RoboDK station: Proyecto_Puhueyestewa_Espinoza.rdk

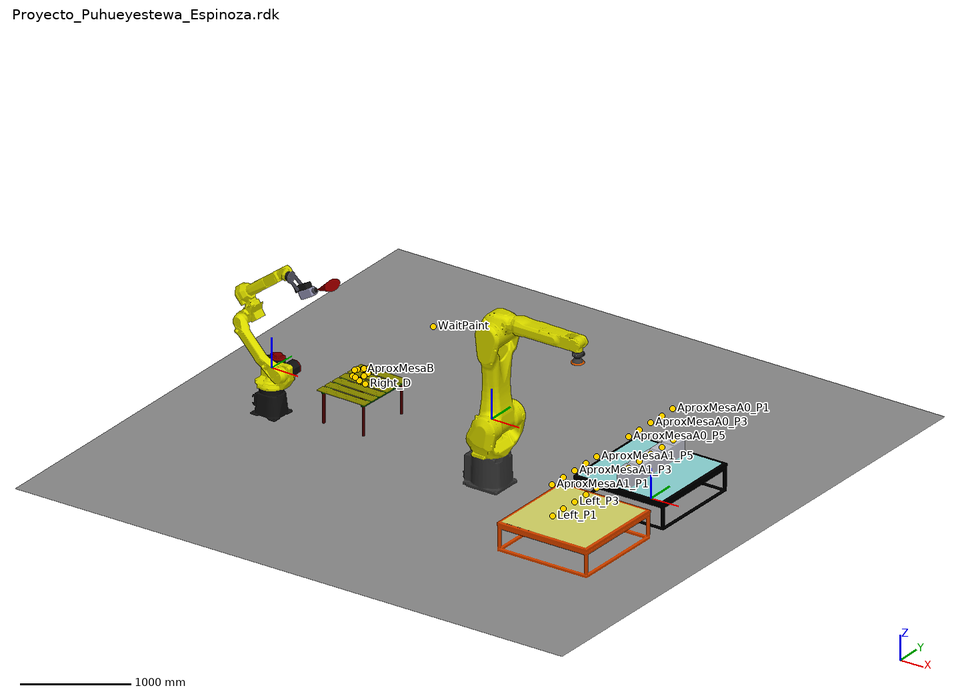
[picture v0: the station drawn from its stored meshes, robots at their saved joint values, targets as dots, program paths as lines]
Station Proyecto_Puhueyestewa_Espinoza (saved by RoboDK 5.3.0). Poses are relative to the parent item; angles as X-Y-Z fixed-axis rotations.
Station parameters (name, value as stored): ColorObject, 3
  - object MesaA1 at (3000, -2200, 0) mm, size 985.8 x 1004.9 x 291.9 mm, geometry from Table-108x114x32-IN.sld
  - object MesaB at (259.9, -1602.19, 600) mm, rotated rx 0 ry 0 rz 88.1 deg, size 656.6 x 530.9 x 335.3 mm, geometry from welding_table.sld
  - frame RobotA Base at (1676.97, -1606.48, 650) mm
    - robot RobotA (model Fanuc M-20iB/25): 6 axes, payload 25 kg, reach 1853 mm, repeatability 0.05 mm, weight 210 kg
        modified DH rows (alpha deg, a mm, theta deg, d mm): 0, 0, 0, 650; -90, 80, -90, 0; 0, 905, 0, 0; -90, 120, 0, 865; 90, 0, 0, 0; -90, 0, 0, 100
        base shift (0, 0, -650) mm
        joint limits [-180, -120, -70, -200, -145, -270] to [180, 120, 230, 200, 145, 270]; home [0, 0, 0, 0, -90, 0]; saved at [0, 0, 0, 0, -90, 180]
      - tool RobotiQ Sanding Kit, TCP at (0, 0, 90.86) mm, size 127 x 139.7 x 103.3 mm
    - target AproxMesaA0_P1 (Cartesian target) at (1323.03, 955.18, 93.07) mm, rotated rx 180 ry 0 rz 0 deg; joints [35.828, 52.673, -25.551, 0, -64.449, -35.828] of RobotA
    - target AproxMesaA0_P2 (Cartesian target) at (1323.03, 780.66, 93.07) mm, rotated rx 180 ry 0 rz 0 deg; joints [30.543, 46.178, -31.005, 0, -58.995, -30.543] of RobotA
    - target AproxMesaA0_P3 (Cartesian target) at (1323.03, 606.48, 93.07) mm, rotated rx -180 ry 0 rz 0 deg; joints [24.627, 41.286, -34.872, 0, -55.128, -24.627] of RobotA
    - target AproxMesaA0_P4 (Cartesian target) at (1323.03, 430.87, 93.07) mm, rotated rx -180 ry 0 rz 0 deg; joints [18.039, 37.651, -37.592, 0, -52.408, -18.039] of RobotA
    - target AproxMesaA0_P5 (Cartesian target) at (1323.03, 257.29, 93.07) mm, rotated rx -180 ry 0 rz 0 deg; joints [11.005, 35.26, -39.302, 0, -50.698, -11.005] of RobotA
    - target AproxMesaA1_P1 (Cartesian target) at (1323.03, -935.11, 93.07) mm, rotated rx -180 ry 0 rz 0 deg; joints [-35.252, 51.823, -26.284, 0, -63.716, 35.252] of RobotA
    - target AproxMesaA1_P2 (Cartesian target) at (1323.03, -761.53, 93.07) mm, rotated rx -180 ry 0 rz 0 deg; joints [-29.925, 45.572, -31.496, 0, -58.504, 29.925] of RobotA
    - target AproxMesaA1_P3 (Cartesian target) at (1323.03, -585.91, 93.07) mm, rotated rx -180 ry 0 rz 0 deg; joints [-23.886, 40.795, -35.247, 0, -54.753, 23.886] of RobotA
    - target AproxMesaA1_P4 (Cartesian target) at (1323.03, -411.74, 93.07) mm, rotated rx -180 ry 0 rz 0 deg; joints [-17.287, 37.329, -37.826, 0, -52.174, 17.287] of RobotA
    - target AproxMesaA1_P5 (Cartesian target) at (1323.03, -237.21, 93.07) mm, rotated rx -180 ry 0 rz 0 deg; joints [-10.165, 35.061, -39.441, 0, -50.559, 10.165] of RobotA
    - target Take_P1 (Cartesian target) at (1323.03, 956.48, -220.35) mm, rotated rx -180 ry 0 rz 0 deg; joints [35.865, 62.489, -38.726, 0, -51.274, -35.865] of RobotA
    - target Take_P2 (Cartesian target) at (1323.03, 780.66, -220.35) mm, rotated rx -180 ry 0 rz 0 deg; joints [30.543, 56.858, -44.792, 0, -45.208, -30.543] of RobotA
    - target Take_P3 (Cartesian target) at (1323.03, 606.48, -220.35) mm, rotated rx -180 ry 0 rz 0 deg; joints [24.627, 52.739, -49.29, 0, -40.71, -24.627] of RobotA
    - target Take_P4 (Cartesian target) at (1323.03, 430.87, -220.35) mm, rotated rx -180 ry 0 rz 0 deg; joints [18.039, 49.747, -52.598, 0, -37.402, -18.039] of RobotA
    - target Take_P5 (Cartesian target) at (1323.03, 257.29, -220.35) mm, rotated rx -180 ry 0 rz 0 deg; joints [11.005, 47.819, -54.753, 0, -35.247, -11.005] of RobotA
    - target Left_P1 (Cartesian target) at (1323.03, -933.81, -220.35) mm, rotated rx -180 ry 0 rz 0 deg; joints [-35.215, 61.659, -39.615, 0, -50.385, 35.215] of RobotA
    - target Left_P2 (Cartesian target) at (1323.03, -760.23, -220.35) mm, rotated rx -180 ry 0 rz 0 deg; joints [-29.882, 56.308, -45.389, 0, -44.611, 29.882] of RobotA
    - target Left_P3 (Cartesian target) at (1323.03, -584.61, -220.35) mm, rotated rx -180 ry 0 rz 0 deg; joints [-23.839, 52.306, -49.766, 0, -40.234, 23.839] of RobotA
    - target Left_P4 (Cartesian target) at (1323.03, -410.44, -220.35) mm, rotated rx -180 ry 0 rz 0 deg; joints [-17.235, 49.468, -52.909, 0, -37.091, 17.235] of RobotA
    - target Left_P5 (Cartesian target) at (1323.03, -235.91, -220.35) mm, rotated rx -180 ry 0 rz 0 deg; joints [-10.11, 47.649, -54.944, 0, -35.056, 10.11] of RobotA
    - target AproxMesaB (Cartesian target) at (-1417.07, 4.29, 103.23) mm, rotated rx 180 ry 0 rz 0 deg; joints [179.826, 38.777, -36.006, 0, -53.994, -179.826] of RobotA
    - target WaitPaint (Cartesian target) at (-643.02, 4.29, 741.53) mm, rotated rx 180 ry 0 rz 0 deg; joints [179.617, -20.046, -8.465, 0, -81.535, -179.617] of RobotA
    - frame MesaA0 Base at (1323.03, 606.48, -660.35) mm
      - object MesaA0 at (0, 0, 0) mm, size 985.8 x 1004.9 x 291.9 mm, geometry from Table-108x114x32-IN.sld
  - frame RobotB Base at (-785.52, -1535.25, 450) mm, rotated rx 0 ry 0 rz -3 deg
    - robot RobotB (model Fanuc M-10iA): 6 axes, payload 10 kg, reach 1420 mm, repeatability 0.08 mm, weight 130 kg
        modified DH rows (alpha deg, a mm, theta deg, d mm): 0, 0, 0, 450; -90, 150, -90, 0; 0, 600, 0, 0; -90, 200, 0, 640; 90, 0, 0, 0; -90, 0, 0, 100
        base shift (0, 0, -450) mm
        joint limits [-180, -90, -95, -190, -190, -360] to [180, 160, 180, 190, 190, 360]; home [0, -44.52, 36.95, 0, -36.95, 0]; saved at [0, -44.52, 36.95, 180, 36.95, 180]
      - tool Paint gun, TCP at (50, 0, 450) mm, rotated rx 0 ry 30 rz 0 deg, size 203.2 x 279.7 x 471.5 mm
    - target Right_D (Cartesian target) at (1128.46, -77.94, 203.78) mm, rotated rx 90 ry -60.18 rz -173.2 deg; joints [-28.769, 42.471, -20.584, -58.905, -97.457, 150.668] of RobotB
    - target Right_M (Cartesian target) at (1071.48, -84.74, 225.06) mm, rotated rx 90 ry -60.18 rz -173.2 deg; joints [-30.393, 36.873, -21.966, -58.048, -98.024, 152.655] of RobotB
    - target Right_U (Cartesian target) at (1002.27, -93, 254.88) mm, rotated rx 90 ry -60.18 rz -173.2 deg; joints [-32.542, 30.646, -22.514, -57, -99.408, 154.203] of RobotB
    - target Center_D (Cartesian target) at (1011.4, -39.87, 300.37) mm, rotated rx 180 ry 0 rz -173.2 deg; joints [-4.924, -0.5, 0.153, -6.683, -60.84, 193.459] of RobotB
    - target Center_M (Cartesian target) at (1050.89, 5.93, 300.37) mm, rotated rx 180 ry 0 rz -173.2 deg; joints [-1.501, 3.048, 0.227, -4.756, -60.572, 189.546] of RobotB
    - target Center_U (Cartesian target) at (1079.26, 49.09, 300.37) mm, rotated rx 180 ry 0 rz -173.2 deg; joints [1.46, 5.834, 0.429, -3.065, -60.572, 186.138] of RobotB
    - target Left_U (Cartesian target) at (1098.26, 69.52, 285.71) mm, rotated rx -90 ry 0 rz -173.2 deg; joints [33.722, 20.618, -41.647, 92.049, -87.698, 138.311] of RobotB
    - target Left_M (Cartesian target) at (1048.72, 63.61, 234.84) mm, rotated rx -90 ry 0 rz -173.2 deg; joints [35.116, 19.049, -47.063, 91.235, -88.851, 132.925] of RobotB
    - target Left_D (Cartesian target) at (1007.9, 58.74, 193.57) mm, rotated rx -90 ry 0 rz -173.2 deg; joints [36.368, 18.195, -51.506, 90.34, -89.729, 128.493] of RobotB
    - target Face_D (Cartesian target) at (972.74, -18.59, 202.79) mm, rotated rx 0 ry -90 rz -173.2 deg; joints [-9.324, -34.09, -22.694, 120.254, 16.17, 246.957] of RobotB
    - target Face_U (Cartesian target) at (973.71, -26.75, 277.71) mm, rotated rx 0 ry -90 rz -173.2 deg; joints [-10.259, -34.141, -16.259, 134.328, 20.806, 232.465] of RobotB
  - Python program Proceso_Industrial (listed below)
  - Python program Estado_Inicial (listed below)
  - object Floor at (1219.35, -1130.77, 0) mm, size 6000 x 6000 x 0 mm, geometry from Floor.sld
  - object Pieza1 at (3000, -650, 429.65) mm, size 150 x 150 x 150 mm, geometry from box.sld
  - object Pieza2 at (3000, -825, 429.65) mm, size 150 x 150 x 150 mm, geometry from box.sld
  - object Pieza3 at (3000, -1000, 429.65) mm, size 150 x 150 x 150 mm, geometry from box.sld
  - object Pieza4 at (3000, -1175, 429.65) mm, size 150 x 150 x 150 mm, geometry from box.sld
  - object Pieza5 at (3000, -1350, 429.65) mm, size 150 x 150 x 150 mm, geometry from box.sld

--- Python program Proceso_Industrial ---
#Laboratorio de Robótica Industrial - Proyecto
#Docente: Ing. María Jose Ramirez Prado
#Integrantes del grupo: Henry Puhueyestewa Sarango - Miguel Espinoza Peña
#Proyecto: Pintado de Objetos
#Paralelo 103

#¬¬¬¬¬¬¬¬¬¬¬¬¬¬¬¬¬¬¬¬¬¬¬¬¬¬¬¬¬¬¬¬¬¬¬¬¬¬¬¬¬¬¬¬¬¬¬¬¬¬¬¬¬¬¬¬¬¬¬¬¬¬¬¬¬¬¬¬¬¬¬¬¬¬¬¬¬¬¬¬¬¬¬¬¬¬¬¬¬¬¬¬¬¬¬¬¬¬¬¬
#ChooseColors¬¬¬¬¬¬¬¬¬¬¬¬¬¬¬¬¬¬¬¬¬¬¬¬¬¬¬¬¬¬¬¬¬¬¬¬¬¬¬¬¬¬¬¬¬¬¬¬¬¬¬¬¬¬¬¬¬¬¬¬¬¬¬¬¬¬¬¬¬¬¬¬¬¬¬¬¬¬¬¬¬¬¬¬¬¬¬¬
#¬¬¬¬¬¬¬¬¬¬¬¬¬¬¬¬¬¬¬¬¬¬¬¬¬¬¬¬¬¬¬¬¬¬¬¬¬¬¬¬¬¬¬¬¬¬¬¬¬¬¬¬¬¬¬¬¬¬¬¬¬¬¬¬¬¬¬¬¬¬¬¬¬¬¬¬¬¬¬¬¬¬¬¬¬¬¬¬¬¬¬¬¬¬¬¬¬¬¬¬
from robolink import *    # API to communicate with RoboDK
from robodk import *      # basic matrix operations

PARAM_COLOR_OBJECT = 'ColorObject'
RDK = Robolink()
color_object = RDK.getParam(PARAM_COLOR_OBJECT)

color_object_input = mbox('Seleccione el color para pintar el objeto: 1. Rojo, 2. Verde, 3. Azul, 4. Rosado', entry=color_object)
if color_object_input:
    RDK.setParam(PARAM_COLOR_OBJECT, color_object_input)
else:
    raise Exception('Operación cancelada por el usuario')

color=int(color_object_input)

#¬¬¬¬¬¬¬¬¬¬¬¬¬¬¬¬¬¬¬¬¬¬¬¬¬¬¬¬¬¬¬¬¬¬¬¬¬¬¬¬¬¬¬¬¬¬¬¬¬¬¬¬¬¬¬¬¬¬¬¬¬¬¬¬¬¬¬¬¬¬¬¬¬¬¬¬¬¬¬¬¬¬¬¬¬¬¬¬¬¬¬¬¬¬¬¬¬¬¬¬
#Asignación de variables y robots¬¬¬¬¬¬¬¬¬¬¬¬¬¬¬¬¬¬¬¬¬¬¬¬¬¬¬¬¬¬¬¬¬¬¬¬¬¬¬¬¬¬¬¬¬¬¬¬¬¬¬¬¬¬¬¬¬¬¬¬¬¬¬¬¬¬¬¬
#¬¬¬¬¬¬¬¬¬¬¬¬¬¬¬¬¬¬¬¬¬¬¬¬¬¬¬¬¬¬¬¬¬¬¬¬¬¬¬¬¬¬¬¬¬¬¬¬¬¬¬¬¬¬¬¬¬¬¬¬¬¬¬¬¬¬¬¬¬¬¬¬¬¬¬¬¬¬¬¬¬¬¬¬¬¬¬¬¬¬¬¬¬¬¬¬¬¬¬¬
#Se asignan variables a los objetos
toola = 'RobotiQ Sanding Kit'
toolb = 'Paint gun'
objecta = 'Pieza1'
objectb = 'Pieza2'
objectc = 'Pieza3'
objectd = 'Pieza4'
objecte = 'Pieza5'
mesa2 = 'MesaB'
mesa3 = 'MesaA1'
gripper1 = RDK.Item(toola, ITEM_TYPE_TOOL)
gripper2 = RDK.Item(toolb, ITEM_TYPE_TOOL)
pi1 = RDK.Item(objecta, ITEM_TYPE_OBJECT)
pi2 = RDK.Item(objectb, ITEM_TYPE_OBJECT)
pi3 = RDK.Item(objectc, ITEM_TYPE_OBJECT)
pi4 = RDK.Item(objectd, ITEM_TYPE_OBJECT)
pi5 = RDK.Item(objecte, ITEM_TYPE_OBJECT)
mesapaint = RDK.Item(mesa2, ITEM_TYPE_OBJECT)
mesafinal = RDK.Item(mesa3, ITEM_TYPE_OBJECT)

#Con respecto a RobotA
robotA = RDK.Item('RobotA',ITEM_TYPE_ROBOT)
if not robotA.Valid():
    quit()
reference = robotA.Parent()
robotA.setPoseFrame(reference)
pose_ref = robotA.Pose()
print(Pose_2_TxyzRxyz(pose_ref))
home_joints = robotA.JointsHome().tolist()

#Con respecto a RobotB
robotB = RDK.Item('RobotB',ITEM_TYPE_ROBOT)
if not robotB.Valid():
    quit()
reference1 = robotB.Parent()
robotB.setPoseFrame(reference1)
pose_ref1 = robotB.Pose()
print(Pose_2_TxyzRxyz(pose_ref1))
home_joints1 = robotB.JointsHome().tolist()

#¬¬¬¬¬¬¬¬¬¬¬¬¬¬¬¬¬¬¬¬¬¬¬¬¬¬¬¬¬¬¬¬¬¬¬¬¬¬¬¬¬¬¬¬¬¬¬¬¬¬¬¬¬¬¬¬¬¬¬¬¬¬¬¬¬¬¬¬¬¬¬¬¬¬¬¬¬¬¬¬¬¬¬¬¬¬¬¬¬¬¬¬¬¬¬¬¬¬¬¬
#Limpio a pintura anterior¬¬¬¬¬¬¬¬¬¬¬¬¬¬¬¬¬¬¬¬¬¬¬¬¬¬¬¬¬¬¬¬¬¬¬¬¬¬¬¬¬¬¬¬¬¬¬¬¬¬¬¬¬¬¬¬¬¬¬¬¬¬¬¬¬¬¬¬¬¬¬¬¬¬¬
#¬¬¬¬¬¬¬¬¬¬¬¬¬¬¬¬¬¬¬¬¬¬¬¬¬¬¬¬¬¬¬¬¬¬¬¬¬¬¬¬¬¬¬¬¬¬¬¬¬¬¬¬¬¬¬¬¬¬¬¬¬¬¬¬¬¬¬¬¬¬¬¬¬¬¬¬¬¬¬¬¬¬¬¬¬¬¬¬¬¬¬¬¬¬¬¬¬¬¬¬
RDK.Spray_Clear()               #Limpio la pintura
pi1.Recolor([0.90,0.91,0.96,1]) #La pieza inicia blanca
pi2.Recolor([0.90,0.91,0.96,1]) #La pieza inicia blanca
pi3.Recolor([0.90,0.91,0.96,1]) #La pieza inicia blanca
pi4.Recolor([0.90,0.91,0.96,1]) #La pieza inicia blanca
pi5.Recolor([0.90,0.91,0.96,1]) #La pieza inicia blanca

#¬¬¬¬¬¬¬¬¬¬¬¬¬¬¬¬¬¬¬¬¬¬¬¬¬¬¬¬¬¬¬¬¬¬¬¬¬¬¬¬¬¬¬¬¬¬¬¬¬¬¬¬¬¬¬¬¬¬¬¬¬¬¬¬¬¬¬¬¬¬¬¬¬¬¬¬¬¬¬¬¬¬¬¬¬¬¬¬¬¬¬¬¬¬¬¬¬¬¬¬
#Process_Pieza1¬¬¬¬¬¬¬¬¬¬¬¬¬¬¬¬¬¬¬¬¬¬¬¬¬¬¬¬¬¬¬¬¬¬¬¬¬¬¬¬¬¬¬¬¬¬¬¬¬¬¬¬¬¬¬¬¬¬¬¬¬¬¬¬¬¬¬¬¬¬¬¬¬¬¬¬¬¬¬¬¬¬¬¬¬¬
#¬¬¬¬¬¬¬¬¬¬¬¬¬¬¬¬¬¬¬¬¬¬¬¬¬¬¬¬¬¬¬¬¬¬¬¬¬¬¬¬¬¬¬¬¬¬¬¬¬¬¬¬¬¬¬¬¬¬¬¬¬¬¬¬¬¬¬¬¬¬¬¬¬¬¬¬¬¬¬¬¬¬¬¬¬¬¬¬¬¬¬¬¬¬¬¬¬¬¬¬
#Tarea Pick and Place en area de trabajo A0
#RobotA se aproxima a MesaA0 para recoger la pieza
aprox=20
a1 = transl(1323.030,955.182,93.068)*roty(pi)
robotA.MoveJ(a1)
robotA.setSpeed(1000)
#RobotA toma la pieza1 de la MesaA0
b1 = transl(1323.030,956.483,-220.350)*roty(pi)
robotA.MoveJ(b1)
robotA.setSpeed(1000)
pi1.setParentStatic(gripper1)
#RobotA lleva la pieza1 cerca de la MesaB
c1=transl(-1417.075,4.293,400.446)*roty(pi)
robotA.MoveJ(c1)
robotA.setSpeed(1000)
#RobotA deja la pieza1 en la MesaB
d1=transl(-1417.075,4.293,100.367)*roty(pi)
robotA.MoveJ(d1)
robotA.setSpeed(1000)
gripper1.DetachAll()
pi1.setParentStatic(mesapaint)
#RobotA se ubica en la posición de espera
e1=transl(-643.019,4.293,741.529)*roty(pi)
robotA.MoveJ(e1)
robotA.setSpeed(1000)
#RobotB se aproxima a MesaB
aprox=20
a02 = xyzrpw_2_pose([951.091,-99.100,515.373,90.000,-60.175,-173.197])
robotB.MoveJ(a02)
robotB.setSpeed(100)

#¬¬¬¬¬¬¬¬¬¬¬¬¬¬¬¬¬¬¬¬¬¬¬¬¬¬¬¬¬¬¬¬¬¬¬¬¬¬¬¬¬¬¬¬¬¬¬¬¬¬¬¬¬¬¬¬¬¬¬¬¬¬¬¬¬¬¬¬¬¬¬¬¬¬¬¬¬¬¬¬¬¬¬¬¬¬¬¬¬¬¬¬¬¬¬¬¬¬¬¬
#SprayOn1¬¬¬¬¬¬¬¬¬¬¬¬¬¬¬¬¬¬¬¬¬¬¬¬¬¬¬¬¬¬¬¬¬¬¬¬¬¬¬¬¬¬¬¬¬¬¬¬¬¬¬¬¬¬¬¬¬¬¬¬¬¬¬¬¬¬¬¬¬¬¬¬¬¬¬¬¬¬¬¬¬¬¬¬¬¬¬¬¬¬¬¬
#¬¬¬¬¬¬¬¬¬¬¬¬¬¬¬¬¬¬¬¬¬¬¬¬¬¬¬¬¬¬¬¬¬¬¬¬¬¬¬¬¬¬¬¬¬¬¬¬¬¬¬¬¬¬¬¬¬¬¬¬¬¬¬¬¬¬¬¬¬¬¬¬¬¬¬¬¬¬¬¬¬¬¬¬¬¬¬¬¬¬¬¬¬¬¬¬¬¬¬¬
Tool_Name = 'Paint gun'
Object_Name = 'Pieza1'

# Define the default action (0 to deactivate, +1 to activate, -1 to clear any spray gun simulation)
# Setting it to None will display a message
ACTION = +1

# quit if we are not in simulation mode
if RDK.RunMode() != RUNMODE_SIMULATE:
    quit()

# Get any previously added spray gun simulations and display statistics (spray on the part vs spray falling out of the part)
info, data = RDK.Spray_GetStats()
if data.size(1) > 0:
    print("Spray gun statistics:")
    print(info)
    print(data.tr())
    RDK.Spray_Clear()

# Check if we are running this program inside another program and passing arguments
import sys
if len(sys.argv) > 1:
    ACTION = int(sys.argv[1])

# If the default ACTION is None, display a message to activate/deactivate the spray gun
if ACTION is None:
    print('Note: This macro can be called as Spray(1) or SprayOn(0)')
    entry = mbox('Turn gun ON or OFF', ('On', '1'), ('Off', '0'))
    if not entry:
        quit()
    ACTION = int(entry)

if ACTION == 0:
    # Turn the gun off
    RDK.Spray_SetState(SPRAY_OFF)

elif ACTION < 0:
    # Clear all spray simulations (same as pressing ESC key)
    RDK.Spray_Clear()

elif ACTION > 0:

    tool = 0    # auto detect active tool
    obj = 0     # auto detect object in active reference frame
    if Tool_Name is not None:
        tool = RDK.Item(Tool_Name, ITEM_TYPE_TOOL)

    if Object_Name is not None:
        obj = RDK.Item(Object_Name, ITEM_TYPE_OBJECT)

    #options_command = "ELLYPSE PROJECT PARTICLE=SPHERE(4,8,1,1,0.5) STEP=8x8 RAND=2" # simulate
    options_command = "PARTICLE=CUBE(10,10,2) STEP=8x8"

    # Another example with a varying rectancular shape
    # define the rectangular volume as p0, pA, pB, colorRGBA (close and far)
    if color == 1:
        close_param = [-90,-117,  0,  90,-117,0,   -90,117,  0,       1,0,0,1]
        far_param   = [-175,-190,200, 175,-190,200,   -175,190,200,   1,0,0,0.2]
        volume = Mat([close_param, far_param])
        RDK.Spray_Add(tool, obj, "RECTANGLE PARTICLE=SPHERE(2,5) STEP=15x15 RAND=3", volume.tr())
        RDK.Spray_SetState(SPRAY_ON)

    if color == 2:
        close_param = [-90,-117,  0,  90,-117,0,   -90,117,  0,       0,1,0,1]
        far_param   = [-175,-190,200, 175,-190,200,   -175,190,200,   1,0,0,0.2]
        volume = Mat([close_param, far_param])
        RDK.Spray_Add(tool, obj, "RECTANGLE PARTICLE=SPHERE(2,5) STEP=15x15 RAND=3", volume.tr())
        RDK.Spray_SetState(SPRAY_ON)

    if color == 3:
        close_param = [-90,-117,  0,  90,-117,0,   -90,117,  0,       0,0,1,1]
        far_param   = [-175,-190,200, 175,-190,200,   -175,190,200,   1,0,0,0.2]
        volume = Mat([close_param, far_param])
        RDK.Spray_Add(tool, obj, "RECTANGLE PARTICLE=SPHERE(2,5) STEP=15x15 RAND=3", volume.tr())
        RDK.Spray_SetState(SPRAY_ON)

    if color == 4:
        close_param = [-90,-117,  0,  90,-117,0,   -90,117,  0,       1,0,1,1]
        far_param   = [-175,-190,200, 175,-190,200,   -175,190,200,   1,0,0,0.2]
        volume = Mat([close_param, far_param])
        RDK.Spray_Add(tool, obj, "RECTANGLE PARTICLE=SPHERE(2,5) STEP=15x15 RAND=3", volume.tr())
        RDK.Spray_SetState(SPRAY_ON)

#¬¬¬¬¬¬¬¬¬¬¬¬¬¬¬¬¬¬¬¬¬¬¬¬¬¬¬¬¬¬¬¬¬¬¬¬¬¬¬¬¬¬¬¬¬¬¬¬¬¬¬¬¬¬¬¬¬¬¬¬¬¬¬¬¬¬¬¬¬¬¬¬¬¬¬¬¬¬¬¬¬¬¬¬¬¬¬¬¬¬¬¬¬¬¬¬¬¬¬¬
#PP1_A¬¬¬¬¬¬¬¬¬¬¬¬¬¬¬¬¬¬¬¬¬¬¬¬¬¬¬¬¬¬¬¬¬¬¬¬¬¬¬¬¬¬¬¬¬¬¬¬¬¬¬¬¬¬¬¬¬¬¬¬¬¬¬¬¬¬¬¬¬¬¬¬¬¬¬¬¬¬¬¬¬¬¬¬¬¬¬¬¬¬¬¬¬¬¬
#¬¬¬¬¬¬¬¬¬¬¬¬¬¬¬¬¬¬¬¬¬¬¬¬¬¬¬¬¬¬¬¬¬¬¬¬¬¬¬¬¬¬¬¬¬¬¬¬¬¬¬¬¬¬¬¬¬¬¬¬¬¬¬¬¬¬¬¬¬¬¬¬¬¬¬¬¬¬¬¬¬¬¬¬¬¬¬¬¬¬¬¬¬¬¬¬¬¬¬¬
#Tarea Pintado en area de trabajo B
#RobotB pinta pieza1, lado derecho
aprox=20
a2 = xyzrpw_2_pose([1128.463,-77.940,203.783,90.000,-60.175,-173.197])
robotB.MoveJ(a2)
robotB.setSpeed(100)
c2 = xyzrpw_2_pose([1071.476,-84.739,225.057,90.000,-60.175,-173.197])
robotB.MoveJ(c2)
robotB.setSpeed(1000)
d2 = xyzrpw_2_pose([1002.267,-92.996,254.878,90.000,-60.175,-173.197])
robotB.MoveJ(d2)
robotB.setSpeed(1000)
#RobotB pinta pieza1, centro
e2 = xyzrpw_2_pose([1011.397,-39.866,300.368,180.000,0.000,-173.197])
robotB.MoveJ(e2)
robotB.setSpeed(1000)
f2 = xyzrpw_2_pose([1050.893,5.934,300.367,180.000,0.000,-173.197])
robotB.MoveJ(f2)
robotB.setSpeed(1000)
g2 = xyzrpw_2_pose([1079.262,49.092,300.367,180.000,0.000,-173.197])
robotB.MoveJ(g2)
robotB.setSpeed(1000)
#RobotB pinta pieza1, lado izquierdo
h2 = xyzrpw_2_pose([1098.260,69.520,285.711,-90.000,0.000,-173.197])
robotB.MoveJ(h2)
robotB.setSpeed(1000)
i2 = xyzrpw_2_pose([1048.722,63.609,234.840,-90.000,0.000,-173.197])
robotB.MoveJ(i2)
robotB.setSpeed(1000)
j2 = xyzrpw_2_pose([1007.902,58.739,193.572,-90.000,0.000,-173.197])
robotB.MoveJ(j2)
robotB.setSpeed(1000)
#RobotB pinta pieza1, frente
k2 = xyzrpw_2_pose([972.738,-18.594,202.789,0.000,-90.000,-173.197])
robotB.MoveJ(k2)
robotB.setSpeed(1000)
l2 = xyzrpw_2_pose([973.710,-26.748,277.710,0.000,-90.000,-173.197])
robotB.MoveJ(l2)
robotB.setSpeed(1000)
#RobotB se mueve a la posición de home
b2 = xyzrpw_2_pose([670.544,0.000,1022.351,0.000,-60.000,-180.000])
robotB.MoveJ(b2)
robotB.setSpeed(100)
#Color
if color == 1:
    pi1.Recolor([1,0,0,1])
if color == 2:
    pi1.Recolor([0,1,0,1])
if color == 3:
    pi1.Recolor([0,0,1,1])
if color == 4:
    pi1.Recolor([1,0,1,1])

#¬¬¬¬¬¬¬¬¬¬¬¬¬¬¬¬¬¬¬¬¬¬¬¬¬¬¬¬¬¬¬¬¬¬¬¬¬¬¬¬¬¬¬¬¬¬¬¬¬¬¬¬¬¬¬¬¬¬¬¬¬¬¬¬¬¬¬¬¬¬¬¬¬¬¬¬¬¬¬¬¬¬¬¬¬¬¬¬¬¬¬¬¬¬¬¬¬¬¬¬
#PP1_B¬¬¬¬¬¬¬¬¬¬¬¬¬¬¬¬¬¬¬¬¬¬¬¬¬¬¬¬¬¬¬¬¬¬¬¬¬¬¬¬¬¬¬¬¬¬¬¬¬¬¬¬¬¬¬¬¬¬¬¬¬¬¬¬¬¬¬¬¬¬¬¬¬¬¬¬¬¬¬¬¬¬¬¬¬¬¬¬¬¬¬¬¬¬¬
#¬¬¬¬¬¬¬¬¬¬¬¬¬¬¬¬¬¬¬¬¬¬¬¬¬¬¬¬¬¬¬¬¬¬¬¬¬¬¬¬¬¬¬¬¬¬¬¬¬¬¬¬¬¬¬¬¬¬¬¬¬¬¬¬¬¬¬¬¬¬¬¬¬¬¬¬¬¬¬¬¬¬¬¬¬¬¬¬¬¬¬¬¬¬¬¬¬¬¬¬
#Tarea Pick and Place en area de trabajo A1
#RobotA toma la pieza1 de la MesaB
a3=transl(-1417.075,4.293,100.367)*roty(pi)
robotA.MoveJ(a3)
robotA.setSpeed(1000)
mesapaint.DetachAll()
pi1.setParentStatic(gripper1)
#RobotA lleva la pieza1 lejos de la MesaB
b3=transl(-1417.075,4.293,400.446)*roty(pi)
robotA.MoveJ(b3)
robotA.setSpeed(1000)
#RobotA lleva la pieza1 entre MesaB y MesaA1
f3=transl(1323.030,955.182,93.068)*roty(pi)
robotA.MoveJ(f3)
robotA.setSpeed(1000)
#RobotA lleva la pieza1 cerca de la MesaA1
c3=transl(1323.030,-935.107,93.068)*roty(pi)
robotA.MoveJ(c3)
robotA.setSpeed(1000)
#RobotA deja la pieza1 en la MesaA1
d3=transl(1323.030,-933.806,-220.350)*roty(pi)
robotA.MoveJ(d3)
robotA.setSpeed(1000)
gripper1.DetachAll()
pi1.setParentStatic(mesafinal)
#RobotA se mueve a la posición de home
e3=transl(945.000,0.000,834.135)*roty(pi)
robotA.MoveJ(e3)
robotA.setSpeed(1000)

#¬¬¬¬¬¬¬¬¬¬¬¬¬¬¬¬¬¬¬¬¬¬¬¬¬¬¬¬¬¬¬¬¬¬¬¬¬¬¬¬¬¬¬¬¬¬¬¬¬¬¬¬¬¬¬¬¬¬¬¬¬¬¬¬¬¬¬¬¬¬¬¬¬¬¬¬¬¬¬¬¬¬¬¬¬¬¬¬¬¬¬¬¬¬¬¬¬¬¬¬
#Process_Pieza2¬¬¬¬¬¬¬¬¬¬¬¬¬¬¬¬¬¬¬¬¬¬¬¬¬¬¬¬¬¬¬¬¬¬¬¬¬¬¬¬¬¬¬¬¬¬¬¬¬¬¬¬¬¬¬¬¬¬¬¬¬¬¬¬¬¬¬¬¬¬¬¬¬¬¬¬¬¬¬¬¬¬¬¬¬¬
#¬¬¬¬¬¬¬¬¬¬¬¬¬¬¬¬¬¬¬¬¬¬¬¬¬¬¬¬¬¬¬¬¬¬¬¬¬¬¬¬¬¬¬¬¬¬¬¬¬¬¬¬¬¬¬¬¬¬¬¬¬¬¬¬¬¬¬¬¬¬¬¬¬¬¬¬¬¬¬¬¬¬¬¬¬¬¬¬¬¬¬¬¬¬¬¬¬¬¬¬
#Tarea Pick and Place en area de trabajo A0
#RobotA se aproxima a MesaA0 para recoger la pieza
aprox=20
a1 = transl(1323.030,780.657,93.068)*roty(pi)      #Se cambia respecto a AproxMesaA0_P________________________
robotA.MoveJ(a1)
robotA.setSpeed(1000)
#RobotA toma la pieza1 de la MesaA0
b1 = transl(1323.030,780.657,-220.350)*roty(pi)    #Se cambia respecto a Take_P________________________
robotA.MoveJ(b1)
robotA.setSpeed(1000)
pi2.setParentStatic(gripper1)                      #Se cambia el pi_____________________________________
#RobotA lleva la pieza1 cerca de la MesaB
c1=transl(-1417.075,4.293,400.446)*roty(pi)
robotA.MoveJ(c1)
robotA.setSpeed(1000)
#RobotA deja la pieza1 en la MesaB
d1=transl(-1417.075,4.293,100.367)*roty(pi)
robotA.MoveJ(d1)
robotA.setSpeed(1000)
gripper1.DetachAll()
pi2.setParentStatic(mesapaint)                     #Se cambia el pi_____________________________________
#RobotA se ubica en la posición de espera
e1=transl(-643.019,4.293,741.529)*roty(pi)
robotA.MoveJ(e1)
robotA.setSpeed(1000)
#RobotB se aproxima a MesaB
aprox=20
a02 = xyzrpw_2_pose([951.091,-99.100,515.373,90.000,-60.175,-173.197])
robotB.MoveJ(a02)
robotB.setSpeed(100)

#¬¬¬¬¬¬¬¬¬¬¬¬¬¬¬¬¬¬¬¬¬¬¬¬¬¬¬¬¬¬¬¬¬¬¬¬¬¬¬¬¬¬¬¬¬¬¬¬¬¬¬¬¬¬¬¬¬¬¬¬¬¬¬¬¬¬¬¬¬¬¬¬¬¬¬¬¬¬¬¬¬¬¬¬¬¬¬¬¬¬¬¬¬¬¬¬¬¬¬¬
#SprayOn2¬¬¬¬¬¬¬¬¬¬¬¬¬¬¬¬¬¬¬¬¬¬¬¬¬¬¬¬¬¬¬¬¬¬¬¬¬¬¬¬¬¬¬¬¬¬¬¬¬¬¬¬¬¬¬¬¬¬¬¬¬¬¬¬¬¬¬¬¬¬¬¬¬¬¬¬¬¬¬¬¬¬¬¬¬¬¬¬¬¬¬¬
#¬¬¬¬¬¬¬¬¬¬¬¬¬¬¬¬¬¬¬¬¬¬¬¬¬¬¬¬¬¬¬¬¬¬¬¬¬¬¬¬¬¬¬¬¬¬¬¬¬¬¬¬¬¬¬¬¬¬¬¬¬¬¬¬¬¬¬¬¬¬¬¬¬¬¬¬¬¬¬¬¬¬¬¬¬¬¬¬¬¬¬¬¬¬¬¬¬¬¬¬
Tool_Name = 'Paint gun'
Object_Name = 'Pieza2'

# Define the default action (0 to deactivate, +1 to activate, -1 to clear any spray gun simulation)
# Setting it to None will display a message
ACTION = +1

# quit if we are not in simulation mode
if RDK.RunMode() != RUNMODE_SIMULATE:
    quit()

# Get any previously added spray gun simulations and display statistics (spray on the part vs spray falling out of the part)
info, data = RDK.Spray_GetStats()
if data.size(1) > 0:
    print("Spray gun statistics:")
    print(info)
    print(data.tr())
    RDK.Spray_Clear()

# Check if we are running this program inside another program and passing arguments
import sys
if len(sys.argv) > 1:
    ACTION = int(sys.argv[1])

# If the default ACTION is None, display a message to activate/deactivate the spray gun
if ACTION is None:
    print('Note: This macro can be called as Spray(1) or SprayOn(0)')
    entry = mbox('Turn gun ON or OFF', ('On', '1'), ('Off', '0'))
    if not entry:
        quit()
    ACTION = int(entry)

if ACTION == 0:
    # Turn the gun off
    RDK.Spray_SetState(SPRAY_OFF)

elif ACTION < 0:
    # Clear all spray simulations (same as pressing ESC key)
    RDK.Spray_Clear()

elif ACTION > 0:

    tool = 0    # auto detect active tool
    obj = 0     # auto detect object in active reference frame
    if Tool_Name is not None:
        tool = RDK.Item(Tool_Name, ITEM_TYPE_TOOL)

    if Object_Name is not None:
        obj = RDK.Item(Object_Name, ITEM_TYPE_OBJECT)

    #options_command = "ELLYPSE PROJECT PARTICLE=SPHERE(4,8,1,1,0.5) STEP=8x8 RAND=2" # simulate
    options_command = "PARTICLE=CUBE(10,10,2) STEP=8x8"

    # Another example with a varying rectancular shape
    # define the rectangular volume as p0, pA, pB, colorRGBA (close and far)
    if color == 1:
        close_param = [-90,-117,  0,  90,-117,0,   -90,117,  0,       1,0,0,1]
        far_param   = [-175,-190,200, 175,-190,200,   -175,190,200,   1,0,0,0.2]
        volume = Mat([close_param, far_param])
        RDK.Spray_Add(tool, obj, "RECTANGLE PARTICLE=SPHERE(2,5) STEP=15x15 RAND=3", volume.tr())
        RDK.Spray_SetState(SPRAY_ON)

    if color == 2:
        close_param = [-90,-117,  0,  90,-117,0,   -90,117,  0,       0,1,0,1]
        far_param   = [-175,-190,200, 175,-190,200,   -175,190,200,   1,0,0,0.2]
        volume = Mat([close_param, far_param])
        RDK.Spray_Add(tool, obj, "RECTANGLE PARTICLE=SPHERE(2,5) STEP=15x15 RAND=3", volume.tr())
        RDK.Spray_SetState(SPRAY_ON)

    if color == 3:
        close_param = [-90,-117,  0,  90,-117,0,   -90,117,  0,       0,0,1,1]
        far_param   = [-175,-190,200, 175,-190,200,   -175,190,200,   1,0,0,0.2]
        volume = Mat([close_param, far_param])
        RDK.Spray_Add(tool, obj, "RECTANGLE PARTICLE=SPHERE(2,5) STEP=15x15 RAND=3", volume.tr())
        RDK.Spray_SetState(SPRAY_ON)

    if color == 4:
        close_param = [-90,-117,  0,  90,-117,0,   -90,117,  0,       1,0,1,1]
        far_param   = [-175,-190,200, 175,-190,200,   -175,190,200,   1,0,0,0.2]
        volume = Mat([close_param, far_param])
        RDK.Spray_Add(tool, obj, "RECTANGLE PARTICLE=SPHERE(2,5) STEP=15x15 RAND=3", volume.tr())
        RDK.Spray_SetState(SPRAY_ON)

#¬¬¬¬¬¬¬¬¬¬¬¬¬¬¬¬¬¬¬¬¬¬¬¬¬¬¬¬¬¬¬¬¬¬¬¬¬¬¬¬¬¬¬¬¬¬¬¬¬¬¬¬¬¬¬¬¬¬¬¬¬¬¬¬¬¬¬¬¬¬¬¬¬¬¬¬¬¬¬¬¬¬¬¬¬¬¬¬¬¬¬¬¬¬¬¬¬¬¬¬
#PP2_A¬¬¬¬¬¬¬¬¬¬¬¬¬¬¬¬¬¬¬¬¬¬¬¬¬¬¬¬¬¬¬¬¬¬¬¬¬¬¬¬¬¬¬¬¬¬¬¬¬¬¬¬¬¬¬¬¬¬¬¬¬¬¬¬¬¬¬¬¬¬¬¬¬¬¬¬¬¬¬¬¬¬¬¬¬¬¬¬¬¬¬¬¬¬¬
#¬¬¬¬¬¬¬¬¬¬¬¬¬¬¬¬¬¬¬¬¬¬¬¬¬¬¬¬¬¬¬¬¬¬¬¬¬¬¬¬¬¬¬¬¬¬¬¬¬¬¬¬¬¬¬¬¬¬¬¬¬¬¬¬¬¬¬¬¬¬¬¬¬¬¬¬¬¬¬¬¬¬¬¬¬¬¬¬¬¬¬¬¬¬¬¬¬¬¬¬
#Tarea Pintado en area de trabajo B
#RobotB pinta pieza1, lado derecho
aprox=20
a2 = xyzrpw_2_pose([1128.463,-77.940,203.783,90.000,-60.175,-173.197])
robotB.MoveJ(a2)
robotB.setSpeed(100)
c2 = xyzrpw_2_pose([1071.476,-84.739,225.057,90.000,-60.175,-173.197])
robotB.MoveJ(c2)
robotB.setSpeed(1000)
d2 = xyzrpw_2_pose([1002.267,-92.996,254.878,90.000,-60.175,-173.197])
robotB.MoveJ(d2)
robotB.setSpeed(1000)
#RobotB pinta pieza1, centro
e2 = xyzrpw_2_pose([1011.397,-39.866,300.368,180.000,0.000,-173.197])
robotB.MoveJ(e2)
robotB.setSpeed(1000)
f2 = xyzrpw_2_pose([1050.893,5.934,300.367,180.000,0.000,-173.197])
robotB.MoveJ(f2)
robotB.setSpeed(1000)
g2 = xyzrpw_2_pose([1079.262,49.092,300.367,180.000,0.000,-173.197])
robotB.MoveJ(g2)
robotB.setSpeed(1000)
#RobotB pinta pieza1, lado izquierdo
h2 = xyzrpw_2_pose([1098.260,69.520,285.711,-90.000,0.000,-173.197])
robotB.MoveJ(h2)
robotB.setSpeed(1000)
i2 = xyzrpw_2_pose([1048.722,63.609,234.840,-90.000,0.000,-173.197])
robotB.MoveJ(i2)
robotB.setSpeed(1000)
j2 = xyzrpw_2_pose([1007.902,58.739,193.572,-90.000,0.000,-173.197])
robotB.MoveJ(j2)
robotB.setSpeed(1000)
#RobotB pinta pieza1, frente
k2 = xyzrpw_2_pose([972.738,-18.594,202.789,0.000,-90.000,-173.197])
robotB.MoveJ(k2)
robotB.setSpeed(1000)
l2 = xyzrpw_2_pose([973.710,-26.748,277.710,0.000,-90.000,-173.197])
robotB.MoveJ(l2)
robotB.setSpeed(1000)
#RobotB se mueve a la posición de home
b2 = xyzrpw_2_pose([670.544,0.000,1022.351,0.000,-60.000,-180.000])
robotB.MoveJ(b2)
robotB.setSpeed(100)
#Color
if color == 1:
    pi2.Recolor([1,0,0,1])
if color == 2:
    pi2.Recolor([0,1,0,1])
if color == 3:
    pi2.Recolor([0,0,1,1])
if color == 4:
    pi2.Recolor([1,0,1,1])

#¬¬¬¬¬¬¬¬¬¬¬¬¬¬¬¬¬¬¬¬¬¬¬¬¬¬¬¬¬¬¬¬¬¬¬¬¬¬¬¬¬¬¬¬¬¬¬¬¬¬¬¬¬¬¬¬¬¬¬¬¬¬¬¬¬¬¬¬¬¬¬¬¬¬¬¬¬¬¬¬¬¬¬¬¬¬¬¬¬¬¬¬¬¬¬¬¬¬¬¬
#PP2_B¬¬¬¬¬¬¬¬¬¬¬¬¬¬¬¬¬¬¬¬¬¬¬¬¬¬¬¬¬¬¬¬¬¬¬¬¬¬¬¬¬¬¬¬¬¬¬¬¬¬¬¬¬¬¬¬¬¬¬¬¬¬¬¬¬¬¬¬¬¬¬¬¬¬¬¬¬¬¬¬¬¬¬¬¬¬¬¬¬¬¬¬¬¬¬
#¬¬¬¬¬¬¬¬¬¬¬¬¬¬¬¬¬¬¬¬¬¬¬¬¬¬¬¬¬¬¬¬¬¬¬¬¬¬¬¬¬¬¬¬¬¬¬¬¬¬¬¬¬¬¬¬¬¬¬¬¬¬¬¬¬¬¬¬¬¬¬¬¬¬¬¬¬¬¬¬¬¬¬¬¬¬¬¬¬¬¬¬¬¬¬¬¬¬¬¬
#Tarea Pick and Place en area de trabajo A1
#RobotA toma la pieza1 de la MesaB
a3=transl(-1417.075,4.293,100.367)*roty(pi)
robotA.MoveJ(a3)
robotA.setSpeed(1000)
mesapaint.DetachAll()
pi2.setParentStatic(gripper1)                          #Se cambia el pi_____________________________________
#RobotA lleva la pieza1 lejos de la MesaB
b3=transl(-1417.075,4.293,400.446)*roty(pi)
robotA.MoveJ(b3)
robotA.setSpeed(1000)
#RobotA lleva la pieza1 entre MesaB y MesaA1
f3=transl(1323.030,780.657,93.068)*roty(pi)            #Se cambia el AproxMesaA0_P_____________________________________
robotA.MoveJ(f3)
robotA.setSpeed(1000)
#RobotA lleva la pieza1 cerca de la MesaA1
c3=transl(1323.030,-761.529,93.068)*roty(pi)           #Se cambia el AproxMesaA1_P__________________________
robotA.MoveJ(c3)
robotA.setSpeed(1000)
#RobotA deja la pieza1 en la MesaA1
d3=transl(1323.030,-760.228,-220.350)*roty(pi)        #Se cambia respecto a Left_P________________________
robotA.MoveJ(d3)
robotA.setSpeed(1000)
gripper1.DetachAll()
pi2.setParentStatic(mesafinal)                        #Se cambia el pi_____________________________________
#RobotA se mueve a la posición de home
e3=transl(945.000,0.000,834.135)*roty(pi)
robotA.MoveJ(e3)
robotA.setSpeed(1000)

#¬¬¬¬¬¬¬¬¬¬¬¬¬¬¬¬¬¬¬¬¬¬¬¬¬¬¬¬¬¬¬¬¬¬¬¬¬¬¬¬¬¬¬¬¬¬¬¬¬¬¬¬¬¬¬¬¬¬¬¬¬¬¬¬¬¬¬¬¬¬¬¬¬¬¬¬¬¬¬¬¬¬¬¬¬¬¬¬¬¬¬¬¬¬¬¬¬¬¬¬
#Process_Pieza3¬¬¬¬¬¬¬¬¬¬¬¬¬¬¬¬¬¬¬¬¬¬¬¬¬¬¬¬¬¬¬¬¬¬¬¬¬¬¬¬¬¬¬¬¬¬¬¬¬¬¬¬¬¬¬¬¬¬¬¬¬¬¬¬¬¬¬¬¬¬¬¬¬¬¬¬¬¬¬¬¬¬¬¬¬¬
#¬¬¬¬¬¬¬¬¬¬¬¬¬¬¬¬¬¬¬¬¬¬¬¬¬¬¬¬¬¬¬¬¬¬¬¬¬¬¬¬¬¬¬¬¬¬¬¬¬¬¬¬¬¬¬¬¬¬¬¬¬¬¬¬¬¬¬¬¬¬¬¬¬¬¬¬¬¬¬¬¬¬¬¬¬¬¬¬¬¬¬¬¬¬¬¬¬¬¬¬
#Tarea Pick and Place en area de trabajo A0
#RobotA se aproxima a MesaA0 para recoger la pieza
aprox=20
a1 = transl(1323.030,606.483,93.068)*roty(pi)      #Se cambia respecto a AproxMesaA0_P________________________
robotA.MoveJ(a1)
robotA.setSpeed(1000)
#RobotA toma la pieza1 de la MesaA0
b1 = transl(1323.030,606.483,-220.350)*roty(pi)    #Se cambia respecto a Take_P________________________
robotA.MoveJ(b1)
robotA.setSpeed(1000)
pi3.setParentStatic(gripper1)                      #Se cambia el pi_____________________________________
#RobotA lleva la pieza1 cerca de la MesaB
c1=transl(-1417.075,4.293,400.446)*roty(pi)
robotA.MoveJ(c1)
robotA.setSpeed(1000)
#RobotA deja la pieza1 en la MesaB
d1=transl(-1417.075,4.293,100.367)*roty(pi)
robotA.MoveJ(d1)
robotA.setSpeed(1000)
gripper1.DetachAll()
pi3.setParentStatic(mesapaint)                     #Se cambia el pi_____________________________________
#RobotA se ubica en la posición de espera
e1=transl(-643.019,4.293,741.529)*roty(pi)
robotA.MoveJ(e1)
robotA.setSpeed(1000)
#RobotB se aproxima a MesaB
aprox=20
a02 = xyzrpw_2_pose([951.091,-99.100,515.373,90.000,-60.175,-173.197])
robotB.MoveJ(a02)
robotB.setSpeed(100)

#¬¬¬¬¬¬¬¬¬¬¬¬¬¬¬¬¬¬¬¬¬¬¬¬¬¬¬¬¬¬¬¬¬¬¬¬¬¬¬¬¬¬¬¬¬¬¬¬¬¬¬¬¬¬¬¬¬¬¬¬¬¬¬¬¬¬¬¬¬¬¬¬¬¬¬¬¬¬¬¬¬¬¬¬¬¬¬¬¬¬¬¬¬¬¬¬¬¬¬¬
#SprayOn3¬¬¬¬¬¬¬¬¬¬¬¬¬¬¬¬¬¬¬¬¬¬¬¬¬¬¬¬¬¬¬¬¬¬¬¬¬¬¬¬¬¬¬¬¬¬¬¬¬¬¬¬¬¬¬¬¬¬¬¬¬¬¬¬¬¬¬¬¬¬¬¬¬¬¬¬¬¬¬¬¬¬¬¬¬¬¬¬¬¬¬¬
#¬¬¬¬¬¬¬¬¬¬¬¬¬¬¬¬¬¬¬¬¬¬¬¬¬¬¬¬¬¬¬¬¬¬¬¬¬¬¬¬¬¬¬¬¬¬¬¬¬¬¬¬¬¬¬¬¬¬¬¬¬¬¬¬¬¬¬¬¬¬¬¬¬¬¬¬¬¬¬¬¬¬¬¬¬¬¬¬¬¬¬¬¬¬¬¬¬¬¬¬
Tool_Name = 'Paint gun'
Object_Name = 'Pieza3'

# Define the default action (0 to deactivate, +1 to activate, -1 to clear any spray gun simulation)
# Setting it to None will display a message
ACTION = +1

# quit if we are not in simulation mode
if RDK.RunMode() != RUNMODE_SIMULATE:
    quit()

# Get any previously added spray gun simulations and display statistics (spray on the part vs spray falling out of the part)
info, data = RDK.Spray_GetStats()
if data.size(1) > 0:
    print("Spray gun statistics:")
    print(info)
    print(data.tr())
    RDK.Spray_Clear()

# Check if we are running this program inside another program and passing arguments
import sys
if len(sys.argv) > 1:
    ACTION = int(sys.argv[1])

# If the default ACTION is None, display a message to activate/deactivate the spray gun
if ACTION is None:
    print('Note: This macro can be called as Spray(1) or SprayOn(0)')
    entry = mbox('Turn gun ON or OFF', ('On', '1'), ('Off', '0'))
    if not entry:
        quit()
    ACTION = int(entry)

if ACTION == 0:
    # Turn the gun off
    RDK.Spray_SetState(SPRAY_OFF)

elif ACTION < 0:
    # Clear all spray simulations (same as pressing ESC key)
    RDK.Spray_Clear()

elif ACTION > 0:

    tool = 0    # auto detect active tool
    obj = 0     # auto detect object in active reference frame
    if Tool_Name is not None:
        tool = RDK.Item(Tool_Name, ITEM_TYPE_TOOL)

    if Object_Name is not None:
        obj = RDK.Item(Object_Name, ITEM_TYPE_OBJECT)

    #options_command = "ELLYPSE PROJECT PARTICLE=SPHERE(4,8,1,1,0.5) STEP=8x8 RAND=2" # simulate
    options_command = "PARTICLE=CUBE(10,10,2) STEP=8x8"

    # Another example with a varying rectancular shape
    # define the rectangular volume as p0, pA, pB, colorRGBA (close and far)
    if color == 1:
        close_param = [-90,-117,  0,  90,-117,0,   -90,117,  0,       1,0,0,1]
        far_param   = [-175,-190,200, 175,-190,200,   -175,190,200,   1,0,0,0.2]
        volume = Mat([close_param, far_param])
        RDK.Spray_Add(tool, obj, "RECTANGLE PARTICLE=SPHERE(2,5) STEP=15x15 RAND=3", volume.tr())
        RDK.Spray_SetState(SPRAY_ON)

    if color == 2:
        close_param = [-90,-117,  0,  90,-117,0,   -90,117,  0,       0,1,0,1]
        far_param   = [-175,-190,200, 175,-190,200,   -175,190,200,   1,0,0,0.2]
        volume = Mat([close_param, far_param])
        RDK.Spray_Add(tool, obj, "RECTANGLE PARTICLE=SPHERE(2,5) STEP=15x15 RAND=3", volume.tr())
        RDK.Spray_SetState(SPRAY_ON)

    if color == 3:
        close_param = [-90,-117,  0,  90,-117,0,   -90,117,  0,       0,0,1,1]
        far_param   = [-175,-190,200, 175,-190,200,   -175,190,200,   1,0,0,0.2]
        volume = Mat([close_param, far_param])
        RDK.Spray_Add(tool, obj, "RECTANGLE PARTICLE=SPHERE(2,5) STEP=15x15 RAND=3", volume.tr())
        RDK.Spray_SetState(SPRAY_ON)

    if color == 4:
        close_param = [-90,-117,  0,  90,-117,0,   -90,117,  0,       1,0,1,1]
        far_param   = [-175,-190,200, 175,-190,200,   -175,190,200,   1,0,0,0.2]
        volume = Mat([close_param, far_param])
        RDK.Spray_Add(tool, obj, "RECTANGLE PARTICLE=SPHERE(2,5) STEP=15x15 RAND=3", volume.tr())
        RDK.Spray_SetState(SPRAY_ON)

#¬¬¬¬¬¬¬¬¬¬¬¬¬¬¬¬¬¬¬¬¬¬¬¬¬¬¬¬¬¬¬¬¬¬¬¬¬¬¬¬¬¬¬¬¬¬¬¬¬¬¬¬¬¬¬¬¬¬¬¬¬¬¬¬¬¬¬¬¬¬¬¬¬¬¬¬¬¬¬¬¬¬¬¬¬¬¬¬¬¬¬¬¬¬¬¬¬¬¬¬
#PP3_A¬¬¬¬¬¬¬¬¬¬¬¬¬¬¬¬¬¬¬¬¬¬¬¬¬¬¬¬¬¬¬¬¬¬¬¬¬¬¬¬¬¬¬¬¬¬¬¬¬¬¬¬¬¬¬¬¬¬¬¬¬¬¬¬¬¬¬¬¬¬¬¬¬¬¬¬¬¬¬¬¬¬¬¬¬¬¬¬¬¬¬¬¬¬¬
#¬¬¬¬¬¬¬¬¬¬¬¬¬¬¬¬¬¬¬¬¬¬¬¬¬¬¬¬¬¬¬¬¬¬¬¬¬¬¬¬¬¬¬¬¬¬¬¬¬¬¬¬¬¬¬¬¬¬¬¬¬¬¬¬¬¬¬¬¬¬¬¬¬¬¬¬¬¬¬¬¬¬¬¬¬¬¬¬¬¬¬¬¬¬¬¬¬¬¬¬
#Tarea Pintado en area de trabajo B
#RobotB pinta pieza1, lado derecho
aprox=20
a2 = xyzrpw_2_pose([1128.463,-77.940,203.783,90.000,-60.175,-173.197])
robotB.MoveJ(a2)
robotB.setSpeed(100)
c2 = xyzrpw_2_pose([1071.476,-84.739,225.057,90.000,-60.175,-173.197])
robotB.MoveJ(c2)
robotB.setSpeed(1000)
d2 = xyzrpw_2_pose([1002.267,-92.996,254.878,90.000,-60.175,-173.197])
robotB.MoveJ(d2)
robotB.setSpeed(1000)
#RobotB pinta pieza1, centro
e2 = xyzrpw_2_pose([1011.397,-39.866,300.368,180.000,0.000,-173.197])
robotB.MoveJ(e2)
robotB.setSpeed(1000)
f2 = xyzrpw_2_pose([1050.893,5.934,300.367,180.000,0.000,-173.197])
robotB.MoveJ(f2)
robotB.setSpeed(1000)
g2 = xyzrpw_2_pose([1079.262,49.092,300.367,180.000,0.000,-173.197])
robotB.MoveJ(g2)
robotB.setSpeed(1000)
#RobotB pinta pieza1, lado izquierdo
h2 = xyzrpw_2_pose([1098.260,69.520,285.711,-90.000,0.000,-173.197])
robotB.MoveJ(h2)
robotB.setSpeed(1000)
i2 = xyzrpw_2_pose([1048.722,63.609,234.840,-90.000,0.000,-173.197])
robotB.MoveJ(i2)
robotB.setSpeed(1000)
j2 = xyzrpw_2_pose([1007.902,58.739,193.572,-90.000,0.000,-173.197])
robotB.MoveJ(j2)
robotB.setSpeed(1000)
#RobotB pinta pieza1, frente
k2 = xyzrpw_2_pose([972.738,-18.594,202.789,0.000,-90.000,-173.197])
robotB.MoveJ(k2)
robotB.setSpeed(1000)
l2 = xyzrpw_2_pose([973.710,-26.748,277.710,0.000,-90.000,-173.197])
robotB.MoveJ(l2)
robotB.setSpeed(1000)
#RobotB se mueve a la posición de home
b2 = xyzrpw_2_pose([670.544,0.000,1022.351,0.000,-60.000,-180.000])
robotB.MoveJ(b2)
robotB.setSpeed(100)
#Color
if color == 1:
    pi3.Recolor([1,0,0,1])
if color == 2:
    pi3.Recolor([0,1,0,1])
if color == 3:
    pi3.Recolor([0,0,1,1])
if color == 4:
    pi3.Recolor([1,0,1,1])

#¬¬¬¬¬¬¬¬¬¬¬¬¬¬¬¬¬¬¬¬¬¬¬¬¬¬¬¬¬¬¬¬¬¬¬¬¬¬¬¬¬¬¬¬¬¬¬¬¬¬¬¬¬¬¬¬¬¬¬¬¬¬¬¬¬¬¬¬¬¬¬¬¬¬¬¬¬¬¬¬¬¬¬¬¬¬¬¬¬¬¬¬¬¬¬¬¬¬¬¬
#PP3_B¬¬¬¬¬¬¬¬¬¬¬¬¬¬¬¬¬¬¬¬¬¬¬¬¬¬¬¬¬¬¬¬¬¬¬¬¬¬¬¬¬¬¬¬¬¬¬¬¬¬¬¬¬¬¬¬¬¬¬¬¬¬¬¬¬¬¬¬¬¬¬¬¬¬¬¬¬¬¬¬¬¬¬¬¬¬¬¬¬¬¬¬¬¬¬
#¬¬¬¬¬¬¬¬¬¬¬¬¬¬¬¬¬¬¬¬¬¬¬¬¬¬¬¬¬¬¬¬¬¬¬¬¬¬¬¬¬¬¬¬¬¬¬¬¬¬¬¬¬¬¬¬¬¬¬¬¬¬¬¬¬¬¬¬¬¬¬¬¬¬¬¬¬¬¬¬¬¬¬¬¬¬¬¬¬¬¬¬¬¬¬¬¬¬¬¬
#Tarea Pick and Place en area de trabajo A1
#RobotA toma la pieza1 de la MesaB
a3=transl(-1417.075,4.293,100.367)*roty(pi)
robotA.MoveJ(a3)
robotA.setSpeed(1000)
mesapaint.DetachAll()
pi3.setParentStatic(gripper1)                          #Se cambia el pi_____________________________________
#RobotA lleva la pieza1 lejos de la MesaB
b3=transl(-1417.075,4.293,400.446)*roty(pi)
robotA.MoveJ(b3)
robotA.setSpeed(1000)
#RobotA lleva la pieza1 entre MesaB y MesaA1
f3=transl(1323.030,606.483,93.068)*roty(pi)            #Se cambia el AproxMesaA0_P_____________________________________
robotA.MoveJ(f3)
robotA.setSpeed(1000)
#RobotA lleva la pieza1 cerca de la MesaA1
c3=transl(1323.030,-585.913,93.068)*roty(pi)           #Se cambia el AproxMesaA1_P__________________________
robotA.MoveJ(c3)
robotA.setSpeed(1000)
#RobotA deja la pieza1 en la MesaA1
d3=transl(1323.030,-584.612,-220.350)*roty(pi)        #Se cambia respecto a Left_P________________________
robotA.MoveJ(d3)
robotA.setSpeed(1000)
gripper1.DetachAll()
pi3.setParentStatic(mesafinal)                        #Se cambia el pi_____________________________________
#RobotA se mueve a la posición de home
e3=transl(945.000,0.000,834.135)*roty(pi)
robotA.MoveJ(e3)
robotA.setSpeed(1000)

#¬¬¬¬¬¬¬¬¬¬¬¬¬¬¬¬¬¬¬¬¬¬¬¬¬¬¬¬¬¬¬¬¬¬¬¬¬¬¬¬¬¬¬¬¬¬¬¬¬¬¬¬¬¬¬¬¬¬¬¬¬¬¬¬¬¬¬¬¬¬¬¬¬¬¬¬¬¬¬¬¬¬¬¬¬¬¬¬¬¬¬¬¬¬¬¬¬¬¬¬
#Process_Pieza4¬¬¬¬¬¬¬¬¬¬¬¬¬¬¬¬¬¬¬¬¬¬¬¬¬¬¬¬¬¬¬¬¬¬¬¬¬¬¬¬¬¬¬¬¬¬¬¬¬¬¬¬¬¬¬¬¬¬¬¬¬¬¬¬¬¬¬¬¬¬¬¬¬¬¬¬¬¬¬¬¬¬¬¬¬¬
#¬¬¬¬¬¬¬¬¬¬¬¬¬¬¬¬¬¬¬¬¬¬¬¬¬¬¬¬¬¬¬¬¬¬¬¬¬¬¬¬¬¬¬¬¬¬¬¬¬¬¬¬¬¬¬¬¬¬¬¬¬¬¬¬¬¬¬¬¬¬¬¬¬¬¬¬¬¬¬¬¬¬¬¬¬¬¬¬¬¬¬¬¬¬¬¬¬¬¬¬
#Tarea Pick and Place en area de trabajo A0
#RobotA se aproxima a MesaA0 para recoger la pieza
aprox=20
a1 = transl(1323.030,430.867,93.068)*roty(pi)      #Se cambia respecto a AproxMesaA0_P________________________
robotA.MoveJ(a1)
robotA.setSpeed(1000)
#RobotA toma la pieza1 de la MesaA0
b1 = transl(1323.030,430.867,-220.350)*roty(pi)    #Se cambia respecto a Take_P________________________
robotA.MoveJ(b1)
robotA.setSpeed(1000)
pi4.setParentStatic(gripper1)                      #Se cambia el pi_____________________________________
#RobotA lleva la pieza1 cerca de la MesaB
c1=transl(-1417.075,4.293,400.446)*roty(pi)
robotA.MoveJ(c1)
robotA.setSpeed(1000)
#RobotA deja la pieza1 en la MesaB
d1=transl(-1417.075,4.293,100.367)*roty(pi)
robotA.MoveJ(d1)
robotA.setSpeed(1000)
gripper1.DetachAll()
pi4.setParentStatic(mesapaint)                     #Se cambia el pi_____________________________________
#RobotA se ubica en la posición de espera
e1=transl(-643.019,4.293,741.529)*roty(pi)
robotA.MoveJ(e1)
robotA.setSpeed(1000)
#RobotB se aproxima a MesaB
aprox=20
a02 = xyzrpw_2_pose([951.091,-99.100,515.373,90.000,-60.175,-173.197])
robotB.MoveJ(a02)
robotB.setSpeed(100)

#¬¬¬¬¬¬¬¬¬¬¬¬¬¬¬¬¬¬¬¬¬¬¬¬¬¬¬¬¬¬¬¬¬¬¬¬¬¬¬¬¬¬¬¬¬¬¬¬¬¬¬¬¬¬¬¬¬¬¬¬¬¬¬¬¬¬¬¬¬¬¬¬¬¬¬¬¬¬¬¬¬¬¬¬¬¬¬¬¬¬¬¬¬¬¬¬¬¬¬¬
#SprayOn4¬¬¬¬¬¬¬¬¬¬¬¬¬¬¬¬¬¬¬¬¬¬¬¬¬¬¬¬¬¬¬¬¬¬¬¬¬¬¬¬¬¬¬¬¬¬¬¬¬¬¬¬¬¬¬¬¬¬¬¬¬¬¬¬¬¬¬¬¬¬¬¬¬¬¬¬¬¬¬¬¬¬¬¬¬¬¬¬¬¬¬¬
#¬¬¬¬¬¬¬¬¬¬¬¬¬¬¬¬¬¬¬¬¬¬¬¬¬¬¬¬¬¬¬¬¬¬¬¬¬¬¬¬¬¬¬¬¬¬¬¬¬¬¬¬¬¬¬¬¬¬¬¬¬¬¬¬¬¬¬¬¬¬¬¬¬¬¬¬¬¬¬¬¬¬¬¬¬¬¬¬¬¬¬¬¬¬¬¬¬¬¬¬
Tool_Name = 'Paint gun'
Object_Name = 'Pieza4'

# Define the default action (0 to deactivate, +1 to activate, -1 to clear any spray gun simulation)
# Setting it to None will display a message
ACTION = +1

# quit if we are not in simulation mode
if RDK.RunMode() != RUNMODE_SIMULATE:
    quit()

# Get any previously added spray gun simulations and display statistics (spray on the part vs spray falling out of the part)
info, data = RDK.Spray_GetStats()
if data.size(1) > 0:
    print("Spray gun statistics:")
    print(info)
    print(data.tr())
    RDK.Spray_Clear()

# Check if we are running this program inside another program and passing arguments
import sys
if len(sys.argv) > 1:
    ACTION = int(sys.argv[1])

# If the default ACTION is None, display a message to activate/deactivate the spray gun
if ACTION is None:
    print('Note: This macro can be called as Spray(1) or SprayOn(0)')
    entry = mbox('Turn gun ON or OFF', ('On', '1'), ('Off', '0'))
    if not entry:
        quit()
    ACTION = int(entry)

if ACTION == 0:
    # Turn the gun off
    RDK.Spray_SetState(SPRAY_OFF)

elif ACTION < 0:
    # Clear all spray simulations (same as pressing ESC key)
    RDK.Spray_Clear()

elif ACTION > 0:

    tool = 0    # auto detect active tool
    obj = 0     # auto detect object in active reference frame
    if Tool_Name is not None:
        tool = RDK.Item(Tool_Name, ITEM_TYPE_TOOL)

    if Object_Name is not None:
        obj = RDK.Item(Object_Name, ITEM_TYPE_OBJECT)

    #options_command = "ELLYPSE PROJECT PARTICLE=SPHERE(4,8,1,1,0.5) STEP=8x8 RAND=2" # simulate
    options_command = "PARTICLE=CUBE(10,10,2) STEP=8x8"

    # Another example with a varying rectancular shape
    # define the rectangular volume as p0, pA, pB, colorRGBA (close and far)
    if color == 1:
        close_param = [-90,-117,  0,  90,-117,0,   -90,117,  0,       1,0,0,1]
        far_param   = [-175,-190,200, 175,-190,200,   -175,190,200,   1,0,0,0.2]
        volume = Mat([close_param, far_param])
        RDK.Spray_Add(tool, obj, "RECTANGLE PARTICLE=SPHERE(2,5) STEP=15x15 RAND=3", volume.tr())
        RDK.Spray_SetState(SPRAY_ON)

    if color == 2:
        close_param = [-90,-117,  0,  90,-117,0,   -90,117,  0,       0,1,0,1]
        far_param   = [-175,-190,200, 175,-190,200,   -175,190,200,   1,0,0,0.2]
        volume = Mat([close_param, far_param])
        RDK.Spray_Add(tool, obj, "RECTANGLE PARTICLE=SPHERE(2,5) STEP=15x15 RAND=3", volume.tr())
        RDK.Spray_SetState(SPRAY_ON)

    if color == 3:
        close_param = [-90,-117,  0,  90,-117,0,   -90,117,  0,       0,0,1,1]
        far_param   = [-175,-190,200, 175,-190,200,   -175,190,200,   1,0,0,0.2]
        volume = Mat([close_param, far_param])
        RDK.Spray_Add(tool, obj, "RECTANGLE PARTICLE=SPHERE(2,5) STEP=15x15 RAND=3", volume.tr())
        RDK.Spray_SetState(SPRAY_ON)

    if color == 4:
        close_param = [-90,-117,  0,  90,-117,0,   -90,117,  0,       1,0,1,1]
        far_param   = [-175,-190,200, 175,-190,200,   -175,190,200,   1,0,0,0.2]
        volume = Mat([close_param, far_param])
        RDK.Spray_Add(tool, obj, "RECTANGLE PARTICLE=SPHERE(2,5) STEP=15x15 RAND=3", volume.tr())
        RDK.Spray_SetState(SPRAY_ON)

#¬¬¬¬¬¬¬¬¬¬¬¬¬¬¬¬¬¬¬¬¬¬¬¬¬¬¬¬¬¬¬¬¬¬¬¬¬¬¬¬¬¬¬¬¬¬¬¬¬¬¬¬¬¬¬¬¬¬¬¬¬¬¬¬¬¬¬¬¬¬¬¬¬¬¬¬¬¬¬¬¬¬¬¬¬¬¬¬¬¬¬¬¬¬¬¬¬¬¬¬
#PP4_A¬¬¬¬¬¬¬¬¬¬¬¬¬¬¬¬¬¬¬¬¬¬¬¬¬¬¬¬¬¬¬¬¬¬¬¬¬¬¬¬¬¬¬¬¬¬¬¬¬¬¬¬¬¬¬¬¬¬¬¬¬¬¬¬¬¬¬¬¬¬¬¬¬¬¬¬¬¬¬¬¬¬¬¬¬¬¬¬¬¬¬¬¬¬¬
#¬¬¬¬¬¬¬¬¬¬¬¬¬¬¬¬¬¬¬¬¬¬¬¬¬¬¬¬¬¬¬¬¬¬¬¬¬¬¬¬¬¬¬¬¬¬¬¬¬¬¬¬¬¬¬¬¬¬¬¬¬¬¬¬¬¬¬¬¬¬¬¬¬¬¬¬¬¬¬¬¬¬¬¬¬¬¬¬¬¬¬¬¬¬¬¬¬¬¬¬
#Tarea Pintado en area de trabajo B
#RobotB pinta pieza1, lado derecho
aprox=20
a2 = xyzrpw_2_pose([1128.463,-77.940,203.783,90.000,-60.175,-173.197])
robotB.MoveJ(a2)
robotB.setSpeed(100)
c2 = xyzrpw_2_pose([1071.476,-84.739,225.057,90.000,-60.175,-173.197])
robotB.MoveJ(c2)
robotB.setSpeed(1000)
d2 = xyzrpw_2_pose([1002.267,-92.996,254.878,90.000,-60.175,-173.197])
robotB.MoveJ(d2)
robotB.setSpeed(1000)
#RobotB pinta pieza1, centro
e2 = xyzrpw_2_pose([1011.397,-39.866,300.368,180.000,0.000,-173.197])
robotB.MoveJ(e2)
robotB.setSpeed(1000)
f2 = xyzrpw_2_pose([1050.893,5.934,300.367,180.000,0.000,-173.197])
robotB.MoveJ(f2)
robotB.setSpeed(1000)
g2 = xyzrpw_2_pose([1079.262,49.092,300.367,180.000,0.000,-173.197])
robotB.MoveJ(g2)
robotB.setSpeed(1000)
#RobotB pinta pieza1, lado izquierdo
h2 = xyzrpw_2_pose([1098.260,69.520,285.711,-90.000,0.000,-173.197])
robotB.MoveJ(h2)
robotB.setSpeed(1000)
i2 = xyzrpw_2_pose([1048.722,63.609,234.840,-90.000,0.000,-173.197])
robotB.MoveJ(i2)
robotB.setSpeed(1000)
j2 = xyzrpw_2_pose([1007.902,58.739,193.572,-90.000,0.000,-173.197])
robotB.MoveJ(j2)
robotB.setSpeed(1000)
#RobotB pinta pieza1, frente
k2 = xyzrpw_2_pose([972.738,-18.594,202.789,0.000,-90.000,-173.197])
robotB.MoveJ(k2)
robotB.setSpeed(1000)
l2 = xyzrpw_2_pose([973.710,-26.748,277.710,0.000,-90.000,-173.197])
robotB.MoveJ(l2)
robotB.setSpeed(1000)
#RobotB se mueve a la posición de home
b2 = xyzrpw_2_pose([670.544,0.000,1022.351,0.000,-60.000,-180.000])
robotB.MoveJ(b2)
robotB.setSpeed(100)
#Color
if color == 1:
    pi4.Recolor([1,0,0,1])
if color == 2:
    pi4.Recolor([0,1,0,1])
if color == 3:
    pi4.Recolor([0,0,1,1])
if color == 4:
    pi4.Recolor([1,0,1,1])

#¬¬¬¬¬¬¬¬¬¬¬¬¬¬¬¬¬¬¬¬¬¬¬¬¬¬¬¬¬¬¬¬¬¬¬¬¬¬¬¬¬¬¬¬¬¬¬¬¬¬¬¬¬¬¬¬¬¬¬¬¬¬¬¬¬¬¬¬¬¬¬¬¬¬¬¬¬¬¬¬¬¬¬¬¬¬¬¬¬¬¬¬¬¬¬¬¬¬¬¬
#PP4_B¬¬¬¬¬¬¬¬¬¬¬¬¬¬¬¬¬¬¬¬¬¬¬¬¬¬¬¬¬¬¬¬¬¬¬¬¬¬¬¬¬¬¬¬¬¬¬¬¬¬¬¬¬¬¬¬¬¬¬¬¬¬¬¬¬¬¬¬¬¬¬¬¬¬¬¬¬¬¬¬¬¬¬¬¬¬¬¬¬¬¬¬¬¬¬
#¬¬¬¬¬¬¬¬¬¬¬¬¬¬¬¬¬¬¬¬¬¬¬¬¬¬¬¬¬¬¬¬¬¬¬¬¬¬¬¬¬¬¬¬¬¬¬¬¬¬¬¬¬¬¬¬¬¬¬¬¬¬¬¬¬¬¬¬¬¬¬¬¬¬¬¬¬¬¬¬¬¬¬¬¬¬¬¬¬¬¬¬¬¬¬¬¬¬¬¬
#Tarea Pick and Place en area de trabajo A1
#RobotA toma la pieza1 de la MesaB
a3=transl(-1417.075,4.293,100.367)*roty(pi)
robotA.MoveJ(a3)
robotA.setSpeed(1000)
mesapaint.DetachAll()
pi4.setParentStatic(gripper1)                          #Se cambia el pi_____________________________________
#RobotA lleva la pieza1 lejos de la MesaB
b3=transl(-1417.075,4.293,400.446)*roty(pi)
robotA.MoveJ(b3)
robotA.setSpeed(1000)
#RobotA lleva la pieza1 entre MesaB y MesaA1
f3=transl(1323.030,430.867,93.068)*roty(pi)            #Se cambia el AproxMesaA0_P_____________________________________
robotA.MoveJ(f3)
robotA.setSpeed(1000)
#RobotA lleva la pieza1 cerca de la MesaA1
c3=transl(1323.030,-411.739,93.068)*roty(pi)           #Se cambia el AproxMesaA1_P__________________________
robotA.MoveJ(c3)
robotA.setSpeed(1000)
#RobotA deja la pieza1 en la MesaA1
d3=transl(1323.030,-410.438,-220.350)*roty(pi)        #Se cambia respecto a Left_P________________________
robotA.MoveJ(d3)
robotA.setSpeed(1000)
gripper1.DetachAll()
pi4.setParentStatic(mesafinal)                        #Se cambia el pi_____________________________________
#RobotA se mueve a la posición de home
e3=transl(945.000,0.000,834.135)*roty(pi)
robotA.MoveJ(e3)
robotA.setSpeed(1000)

#¬¬¬¬¬¬¬¬¬¬¬¬¬¬¬¬¬¬¬¬¬¬¬¬¬¬¬¬¬¬¬¬¬¬¬¬¬¬¬¬¬¬¬¬¬¬¬¬¬¬¬¬¬¬¬¬¬¬¬¬¬¬¬¬¬¬¬¬¬¬¬¬¬¬¬¬¬¬¬¬¬¬¬¬¬¬¬¬¬¬¬¬¬¬¬¬¬¬¬¬
#Process_Pieza5¬¬¬¬¬¬¬¬¬¬¬¬¬¬¬¬¬¬¬¬¬¬¬¬¬¬¬¬¬¬¬¬¬¬¬¬¬¬¬¬¬¬¬¬¬¬¬¬¬¬¬¬¬¬¬¬¬¬¬¬¬¬¬¬¬¬¬¬¬¬¬¬¬¬¬¬¬¬¬¬¬¬¬¬¬¬
#¬¬¬¬¬¬¬¬¬¬¬¬¬¬¬¬¬¬¬¬¬¬¬¬¬¬¬¬¬¬¬¬¬¬¬¬¬¬¬¬¬¬¬¬¬¬¬¬¬¬¬¬¬¬¬¬¬¬¬¬¬¬¬¬¬¬¬¬¬¬¬¬¬¬¬¬¬¬¬¬¬¬¬¬¬¬¬¬¬¬¬¬¬¬¬¬¬¬¬¬
#Tarea Pick and Place en area de trabajo A0
#RobotA se aproxima a MesaA0 para recoger la pieza
aprox=20
a1 = transl(1323.030,257.289,93.068)*roty(pi)      #Se cambia respecto a AproxMesaA0_P________________________
robotA.MoveJ(a1)
robotA.setSpeed(1000)
#RobotA toma la pieza1 de la MesaA0
b1 = transl(1323.030,257.289,-220.350)*roty(pi)    #Se cambia respecto a Take_P________________________
robotA.MoveJ(b1)
robotA.setSpeed(1000)
pi5.setParentStatic(gripper1)                      #Se cambia el pi_____________________________________
#RobotA lleva la pieza1 cerca de la MesaB
c1=transl(-1417.075,4.293,400.446)*roty(pi)
robotA.MoveJ(c1)
robotA.setSpeed(1000)
#RobotA deja la pieza1 en la MesaB
d1=transl(-1417.075,4.293,100.367)*roty(pi)
robotA.MoveJ(d1)
robotA.setSpeed(1000)
gripper1.DetachAll()
pi5.setParentStatic(mesapaint)                     #Se cambia el pi_____________________________________
#RobotA se ubica en la posición de espera
e1=transl(-643.019,4.293,741.529)*roty(pi)
robotA.MoveJ(e1)
robotA.setSpeed(1000)
#RobotB se aproxima a MesaB
aprox=20
a02 = xyzrpw_2_pose([951.091,-99.100,515.373,90.000,-60.175,-173.197])
robotB.MoveJ(a02)
robotB.setSpeed(100)

#¬¬¬¬¬¬¬¬¬¬¬¬¬¬¬¬¬¬¬¬¬¬¬¬¬¬¬¬¬¬¬¬¬¬¬¬¬¬¬¬¬¬¬¬¬¬¬¬¬¬¬¬¬¬¬¬¬¬¬¬¬¬¬¬¬¬¬¬¬¬¬¬¬¬¬¬¬¬¬¬¬¬¬¬¬¬¬¬¬¬¬¬¬¬¬¬¬¬¬¬
#SprayOn5¬¬¬¬¬¬¬¬¬¬¬¬¬¬¬¬¬¬¬¬¬¬¬¬¬¬¬¬¬¬¬¬¬¬¬¬¬¬¬¬¬¬¬¬¬¬¬¬¬¬¬¬¬¬¬¬¬¬¬¬¬¬¬¬¬¬¬¬¬¬¬¬¬¬¬¬¬¬¬¬¬¬¬¬¬¬¬¬¬¬¬¬
#¬¬¬¬¬¬¬¬¬¬¬¬¬¬¬¬¬¬¬¬¬¬¬¬¬¬¬¬¬¬¬¬¬¬¬¬¬¬¬¬¬¬¬¬¬¬¬¬¬¬¬¬¬¬¬¬¬¬¬¬¬¬¬¬¬¬¬¬¬¬¬¬¬¬¬¬¬¬¬¬¬¬¬¬¬¬¬¬¬¬¬¬¬¬¬¬¬¬¬¬
Tool_Name = 'Paint gun'
Object_Name = 'Pieza5'

# Define the default action (0 to deactivate, +1 to activate, -1 to clear any spray gun simulation)
# Setting it to None will display a message
ACTION = +1

# quit if we are not in simulation mode
if RDK.RunMode() != RUNMODE_SIMULATE:
    quit()

# Get any previously added spray gun simulations and display statistics (spray on the part vs spray falling out of the part)
info, data = RDK.Spray_GetStats()
if data.size(1) > 0:
    print("Spray gun statistics:")
    print(info)
    print(data.tr())
    RDK.Spray_Clear()

# Check if we are running this program inside another program and passing arguments
import sys
if len(sys.argv) > 1:
    ACTION = int(sys.argv[1])

# If the default ACTION is None, display a message to activate/deactivate the spray gun
if ACTION is None:
    print('Note: This macro can be called as Spray(1) or SprayOn(0)')
    entry = mbox('Turn gun ON or OFF', ('On', '1'), ('Off', '0'))
    if not entry:
        quit()
    ACTION = int(entry)

if ACTION == 0:
    # Turn the gun off
    RDK.Spray_SetState(SPRAY_OFF)

elif ACTION < 0:
    # Clear all spray simulations (same as pressing ESC key)
    RDK.Spray_Clear()

elif ACTION > 0:

    tool = 0    # auto detect active tool
    obj = 0     # auto detect object in active reference frame
    if Tool_Name is not None:
        tool = RDK.Item(Tool_Name, ITEM_TYPE_TOOL)

    if Object_Name is not None:
        obj = RDK.Item(Object_Name, ITEM_TYPE_OBJECT)

    #options_command = "ELLYPSE PROJECT PARTICLE=SPHERE(4,8,1,1,0.5) STEP=8x8 RAND=2" # simulate
    options_command = "PARTICLE=CUBE(10,10,2) STEP=8x8"

    # Another example with a varying rectancular shape
    # define the rectangular volume as p0, pA, pB, colorRGBA (close and far)
    if color == 1:
        close_param = [-90,-117,  0,  90,-117,0,   -90,117,  0,       1,0,0,1]
        far_param   = [-175,-190,200, 175,-190,200,   -175,190,200,   1,0,0,0.2]
        volume = Mat([close_param, far_param])
        RDK.Spray_Add(tool, obj, "RECTANGLE PARTICLE=SPHERE(2,5) STEP=15x15 RAND=3", volume.tr())
        RDK.Spray_SetState(SPRAY_ON)

    if color == 2:
        close_param = [-90,-117,  0,  90,-117,0,   -90,117,  0,       0,1,0,1]
        far_param   = [-175,-190,200, 175,-190,200,   -175,190,200,   1,0,0,0.2]
        volume = Mat([close_param, far_param])
        RDK.Spray_Add(tool, obj, "RECTANGLE PARTICLE=SPHERE(2,5) STEP=15x15 RAND=3", volume.tr())
        RDK.Spray_SetState(SPRAY_ON)

    if color == 3:
        close_param = [-90,-117,  0,  90,-117,0,   -90,117,  0,       0,0,1,1]
        far_param   = [-175,-190,200, 175,-190,200,   -175,190,200,   1,0,0,0.2]
        volume = Mat([close_param, far_param])
        RDK.Spray_Add(tool, obj, "RECTANGLE PARTICLE=SPHERE(2,5) STEP=15x15 RAND=3", volume.tr())
        RDK.Spray_SetState(SPRAY_ON)

    if color == 4:
        close_param = [-90,-117,  0,  90,-117,0,   -90,117,  0,       1,0,1,1]
        far_param   = [-175,-190,200, 175,-190,200,   -175,190,200,   1,0,0,0.2]
        volume = Mat([close_param, far_param])
        RDK.Spray_Add(tool, obj, "RECTANGLE PARTICLE=SPHERE(2,5) STEP=15x15 RAND=3", volume.tr())
        RDK.Spray_SetState(SPRAY_ON)

#¬¬¬¬¬¬¬¬¬¬¬¬¬¬¬¬¬¬¬¬¬¬¬¬¬¬¬¬¬¬¬¬¬¬¬¬¬¬¬¬¬¬¬¬¬¬¬¬¬¬¬¬¬¬¬¬¬¬¬¬¬¬¬¬¬¬¬¬¬¬¬¬¬¬¬¬¬¬¬¬¬¬¬¬¬¬¬¬¬¬¬¬¬¬¬¬¬¬¬¬
#PP5_A¬¬¬¬¬¬¬¬¬¬¬¬¬¬¬¬¬¬¬¬¬¬¬¬¬¬¬¬¬¬¬¬¬¬¬¬¬¬¬¬¬¬¬¬¬¬¬¬¬¬¬¬¬¬¬¬¬¬¬¬¬¬¬¬¬¬¬¬¬¬¬¬¬¬¬¬¬¬¬¬¬¬¬¬¬¬¬¬¬¬¬¬¬¬¬
#¬¬¬¬¬¬¬¬¬¬¬¬¬¬¬¬¬¬¬¬¬¬¬¬¬¬¬¬¬¬¬¬¬¬¬¬¬¬¬¬¬¬¬¬¬¬¬¬¬¬¬¬¬¬¬¬¬¬¬¬¬¬¬¬¬¬¬¬¬¬¬¬¬¬¬¬¬¬¬¬¬¬¬¬¬¬¬¬¬¬¬¬¬¬¬¬¬¬¬¬
#Tarea Pintado en area de trabajo B
#RobotB pinta pieza1, lado derecho
aprox=20
a2 = xyzrpw_2_pose([1128.463,-77.940,203.783,90.000,-60.175,-173.197])
robotB.MoveJ(a2)
robotB.setSpeed(100)
c2 = xyzrpw_2_pose([1071.476,-84.739,225.057,90.000,-60.175,-173.197])
robotB.MoveJ(c2)
robotB.setSpeed(1000)
d2 = xyzrpw_2_pose([1002.267,-92.996,254.878,90.000,-60.175,-173.197])
robotB.MoveJ(d2)
robotB.setSpeed(1000)
#RobotB pinta pieza1, centro
e2 = xyzrpw_2_pose([1011.397,-39.866,300.368,180.000,0.000,-173.197])
robotB.MoveJ(e2)
robotB.setSpeed(1000)
f2 = xyzrpw_2_pose([1050.893,5.934,300.367,180.000,0.000,-173.197])
robotB.MoveJ(f2)
robotB.setSpeed(1000)
g2 = xyzrpw_2_pose([1079.262,49.092,300.367,180.000,0.000,-173.197])
robotB.MoveJ(g2)
robotB.setSpeed(1000)
#RobotB pinta pieza1, lado izquierdo
h2 = xyzrpw_2_pose([1098.260,69.520,285.711,-90.000,0.000,-173.197])
robotB.MoveJ(h2)
robotB.setSpeed(1000)
i2 = xyzrpw_2_pose([1048.722,63.609,234.840,-90.000,0.000,-173.197])
robotB.MoveJ(i2)
robotB.setSpeed(1000)
j2 = xyzrpw_2_pose([1007.902,58.739,193.572,-90.000,0.000,-173.197])
robotB.MoveJ(j2)
robotB.setSpeed(1000)
#RobotB pinta pieza1, frente
k2 = xyzrpw_2_pose([972.738,-18.594,202.789,0.000,-90.000,-173.197])
robotB.MoveJ(k2)
robotB.setSpeed(1000)
l2 = xyzrpw_2_pose([973.710,-26.748,277.710,0.000,-90.000,-173.197])
robotB.MoveJ(l2)
robotB.setSpeed(1000)
#RobotB se mueve a la posición de home
b2 = xyzrpw_2_pose([670.544,0.000,1022.351,0.000,-60.000,-180.000])
robotB.MoveJ(b2)
robotB.setSpeed(100)
#Color
if color == 1:
    pi5.Recolor([1,0,0,1])
if color == 2:
    pi5.Recolor([0,1,0,1])
if color == 3:
    pi5.Recolor([0,0,1,1])
if color == 4:
    pi5.Recolor([1,0,1,1])

#¬¬¬¬¬¬¬¬¬¬¬¬¬¬¬¬¬¬¬¬¬¬¬¬¬¬¬¬¬¬¬¬¬¬¬¬¬¬¬¬¬¬¬¬¬¬¬¬¬¬¬¬¬¬¬¬¬¬¬¬¬¬¬¬¬¬¬¬¬¬¬¬¬¬¬¬¬¬¬¬¬¬¬¬¬¬¬¬¬¬¬¬¬¬¬¬¬¬¬¬
#PP5_B¬¬¬¬¬¬¬¬¬¬¬¬¬¬¬¬¬¬¬¬¬¬¬¬¬¬¬¬¬¬¬¬¬¬¬¬¬¬¬¬¬¬¬¬¬¬¬¬¬¬¬¬¬¬¬¬¬¬¬¬¬¬¬¬¬¬¬¬¬¬¬¬¬¬¬¬¬¬¬¬¬¬¬¬¬¬¬¬¬¬¬¬¬¬¬
#¬¬¬¬¬¬¬¬¬¬¬¬¬¬¬¬¬¬¬¬¬¬¬¬¬¬¬¬¬¬¬¬¬¬¬¬¬¬¬¬¬¬¬¬¬¬¬¬¬¬¬¬¬¬¬¬¬¬¬¬¬¬¬¬¬¬¬¬¬¬¬¬¬¬¬¬¬¬¬¬¬¬¬¬¬¬¬¬¬¬¬¬¬¬¬¬¬¬¬¬
#Tarea Pick and Place en area de trabajo A1
#RobotA toma la pieza1 de la MesaB
a3=transl(-1417.075,4.293,100.367)*roty(pi)
robotA.MoveJ(a3)
robotA.setSpeed(1000)
mesapaint.DetachAll()
pi5.setParentStatic(gripper1)                          #Se cambia el pi_____________________________________
#RobotA lleva la pieza1 lejos de la MesaB
b3=transl(-1417.075,4.293,400.446)*roty(pi)
robotA.MoveJ(b3)
robotA.setSpeed(1000)
#RobotA lleva la pieza1 entre MesaB y MesaA1
f3=transl(1323.030,257.289,93.068)*roty(pi)            #Se cambia el AproxMesaA0_P_____________________________________
robotA.MoveJ(f3)
robotA.setSpeed(1000)
#RobotA lleva la pieza1 cerca de la MesaA1
c3=transl(1323.030,-237.214,93.068)*roty(pi)           #Se cambia el AproxMesaA1_P__________________________
robotA.MoveJ(c3)
robotA.setSpeed(1000)
#RobotA deja la pieza1 en la MesaA1
d3=transl(1323.030,-235.913,-220.350)*roty(pi)        #Se cambia respecto a Left_P________________________
robotA.MoveJ(d3)
robotA.setSpeed(1000)
gripper1.DetachAll()
pi5.setParentStatic(mesafinal)                        #Se cambia el pi_____________________________________
#RobotA se mueve a la posición de home
e3=transl(945.000,0.000,834.135)*roty(pi)
robotA.MoveJ(e3)
robotA.setSpeed(1000)

--- Python program Estado_Inicial ---
#Laboratorio de Robótica Industrial - Proyecto
#Docente: Ing. María Jose Ramirez Prado
#Integrantes del grupo: Henry Puhueyestewa Sarango - Miguel Espinoza Peña
#Proyecto: Pintado de Objetos
#Paralelo 103


from robolink import *    # API to communicate with RoboDK
from robodk import *      # basic matrix operations
RDK = Robolink()

#¬¬¬¬¬¬¬¬¬¬¬¬¬¬¬¬¬¬¬¬¬¬¬¬¬¬¬¬¬¬¬¬¬¬¬¬¬¬¬¬¬¬¬¬¬¬¬¬¬¬¬¬¬¬¬¬¬¬¬¬¬¬¬¬¬¬¬¬¬¬¬¬¬¬¬¬¬¬¬¬¬¬¬¬¬¬¬¬¬¬¬¬¬¬¬¬¬¬¬¬
#Asignación de variables y robots¬¬¬¬¬¬¬¬¬¬¬¬¬¬¬¬¬¬¬¬¬¬¬¬¬¬¬¬¬¬¬¬¬¬¬¬¬¬¬¬¬¬¬¬¬¬¬¬¬¬¬¬¬¬¬¬¬¬¬¬¬¬¬¬¬¬¬¬
#¬¬¬¬¬¬¬¬¬¬¬¬¬¬¬¬¬¬¬¬¬¬¬¬¬¬¬¬¬¬¬¬¬¬¬¬¬¬¬¬¬¬¬¬¬¬¬¬¬¬¬¬¬¬¬¬¬¬¬¬¬¬¬¬¬¬¬¬¬¬¬¬¬¬¬¬¬¬¬¬¬¬¬¬¬¬¬¬¬¬¬¬¬¬¬¬¬¬¬¬
#Se asignan variables a los objetos
toola = 'RobotiQ Sanding Kit'
toolb = 'Paint gun'
objecta = 'Pieza1'
objectb = 'Pieza2'
objectc = 'Pieza3'
objectd = 'Pieza4'
objecte = 'Pieza5'
mesa2 = 'MesaB'
mesa3 = 'MesaA1'
gripper1 = RDK.Item(toola, ITEM_TYPE_TOOL)
gripper2 = RDK.Item(toolb, ITEM_TYPE_TOOL)
pi1 = RDK.Item(objecta, ITEM_TYPE_OBJECT)
pi2 = RDK.Item(objectb, ITEM_TYPE_OBJECT)
pi3 = RDK.Item(objectc, ITEM_TYPE_OBJECT)
pi4 = RDK.Item(objectd, ITEM_TYPE_OBJECT)
pi5 = RDK.Item(objecte, ITEM_TYPE_OBJECT)
mesapaint = RDK.Item(mesa2, ITEM_TYPE_OBJECT)
mesafinal = RDK.Item(mesa3, ITEM_TYPE_OBJECT)

#Con respecto a RobotA
robotA = RDK.Item('RobotA',ITEM_TYPE_ROBOT)
if not robotA.Valid():
    quit()
reference = robotA.Parent()
robotA.setPoseFrame(reference)
pose_ref = robotA.Pose()
print(Pose_2_TxyzRxyz(pose_ref))
home_joints = robotA.JointsHome().tolist()

#Con respecto a RobotB
robotB = RDK.Item('RobotB',ITEM_TYPE_ROBOT)
if not robotB.Valid():
    quit()
reference1 = robotB.Parent()
robotB.setPoseFrame(reference1)
pose_ref1 = robotB.Pose()
print(Pose_2_TxyzRxyz(pose_ref1))
home_joints1 = robotB.JointsHome().tolist()

#¬¬¬¬¬¬¬¬¬¬¬¬¬¬¬¬¬¬¬¬¬¬¬¬¬¬¬¬¬¬¬¬¬¬¬¬¬¬¬¬¬¬¬¬¬¬¬¬¬¬¬¬¬¬¬¬¬¬¬¬¬¬¬¬¬¬¬¬¬¬¬¬¬¬¬¬¬¬¬¬¬¬¬¬¬¬¬¬¬¬¬¬¬¬¬¬¬¬¬¬
#Limpio la pintura anterior¬¬¬¬¬¬¬¬¬¬¬¬¬¬¬¬¬¬¬¬¬¬¬¬¬¬¬¬¬¬¬¬¬¬¬¬¬¬¬¬¬¬¬¬¬¬¬¬¬¬¬¬¬¬¬¬¬¬¬¬¬¬¬¬¬¬¬¬¬¬¬¬¬¬
#¬¬¬¬¬¬¬¬¬¬¬¬¬¬¬¬¬¬¬¬¬¬¬¬¬¬¬¬¬¬¬¬¬¬¬¬¬¬¬¬¬¬¬¬¬¬¬¬¬¬¬¬¬¬¬¬¬¬¬¬¬¬¬¬¬¬¬¬¬¬¬¬¬¬¬¬¬¬¬¬¬¬¬¬¬¬¬¬¬¬¬¬¬¬¬¬¬¬¬¬
RDK.Spray_Clear()               #Limpio la pintura
pi1.Recolor([0.90,0.91,0.96,1]) #La pieza inicia blanca
pi2.Recolor([0.90,0.91,0.96,1]) #La pieza inicia blanca
pi3.Recolor([0.90,0.91,0.96,1]) #La pieza inicia blanca
pi4.Recolor([0.90,0.91,0.96,1]) #La pieza inicia blanca
pi5.Recolor([0.90,0.91,0.96,1]) #La pieza inicia blanca

#Colocando a posición inicial Pieza1------------------------------------------------------------------
#RobotA se acerca a la MesaA1
ap1=transl(1323.030,-935.107,93.068)*roty(pi)
robotA.MoveJ(ap1)
robotA.setSpeed(1000)
#RobotA toma la pieza1 de la MesaA1
bp1=transl(1323.030,-933.806,-220.350)*roty(pi)
robotA.MoveJ(bp1)
robotA.setSpeed(1000)
mesafinal.DetachAll()
pi1.setParentStatic(gripper1)
#RobotA se aleja de la MesaA1
cp1=transl(1323.030,-935.107,93.068)*roty(pi)
robotA.MoveJ(cp1)
robotA.setSpeed(1000)
#RobotA se aproxima a MesaA0 para dejar la pieza
dp1= transl(1323.030,955.182,93.068)*roty(pi)
robotA.MoveJ(dp1)
robotA.setSpeed(1000)
#RobotA deja la pieza1 en la MesaA0
ep1= transl(1323.030,956.483,-220.350)*roty(pi)
robotA.MoveJ(ep1)
robotA.setSpeed(1000)
gripper1.DetachAll()
#RobotA se mueve a la posición de home
fp1=transl(945.000,0.000,834.135)*roty(pi)
robotA.MoveJ(fp1)
robotA.setSpeed(1000)

#Colocando a posición inicial Pieza2------------------------------------------------------------------
#RobotA se acerca a la MesaA1
ap2=transl(1323.030,-761.529,93.068)*roty(pi)           #Se cambia el AproxMesaA1_P__________________________
robotA.MoveJ(ap2)
robotA.setSpeed(1000)
#RobotA toma la pieza2 de la MesaA1
bp2=transl(1323.030,-760.228,-220.350)*roty(pi)        #Se cambia respecto a Left_P________________________
robotA.MoveJ(bp2)
robotA.setSpeed(1000)
mesafinal.DetachAll()
pi2.setParentStatic(gripper1)                        #Se cambia el pi_____________________________________
#RobotA se aleja de la MesaA1
cp2=transl(1323.030,-761.529,93.068)*roty(pi)           #Se cambia el AproxMesaA1_P__________________________
robotA.MoveJ(cp2)
robotA.setSpeed(1000)
#RobotA se aproxima a MesaA0 para dejar la pieza
dp2= transl(1323.030,780.657,93.068)*roty(pi)      #Se cambia respecto a AproxMesaA0_P________________________
robotA.MoveJ(dp2)
robotA.setSpeed(1000)
#RobotA deja la pieza2 de la MesaA0
ep2= transl(1323.030,780.657,-220.350)*roty(pi)    #Se cambia respecto a Take_P________________________
robotA.MoveJ(ep2)
robotA.setSpeed(1000)
gripper1.DetachAll()                      #Se cambia el pi_____________________________________
#RobotA se mueve a la posición de home
fp2=transl(945.000,0.000,834.135)*roty(pi)
robotA.MoveJ(fp2)
robotA.setSpeed(1000)

#Colocando a posición inicial Pieza3------------------------------------------------------------------
#RobotA se acerca a la MesaA1
ap3=transl(1323.030,-585.913,93.068)*roty(pi)           #Se cambia el AproxMesaA1_P__________________________
robotA.MoveJ(ap3)
robotA.setSpeed(1000)
#RobotA toma la pieza3 de la MesaA1
bp3=transl(1323.030,-584.612,-220.350)*roty(pi)        #Se cambia respecto a Left_P________________________
robotA.MoveJ(bp3)
robotA.setSpeed(1000)
mesafinal.DetachAll()
pi3.setParentStatic(gripper1)                        #Se cambia el pi_____________________________________
#RobotA se aleja de la MesaA1
cp3=transl(1323.030,-585.913,93.068)*roty(pi)           #Se cambia el AproxMesaA1_P__________________________
robotA.MoveJ(cp3)
robotA.setSpeed(1000)
#RobotA se aproxima a MesaA0 para dejar la pieza
dp3= transl(1323.030,606.483,93.068)*roty(pi)      #Se cambia respecto a AproxMesaA0_P________________________
robotA.MoveJ(dp3)
robotA.setSpeed(1000)
#RobotA deja la pieza2 en la MesaA0
ep3= transl(1323.030,606.483,-220.350)*roty(pi)    #Se cambia respecto a Take_P________________________
robotA.MoveJ(ep3)
robotA.setSpeed(1000)
gripper1.DetachAll()                      #Se cambia el pi_____________________________________
#RobotA se mueve a la posición de home
fp3=transl(945.000,0.000,834.135)*roty(pi)
robotA.MoveJ(fp3)
robotA.setSpeed(1000)

#Colocando a posición inicial Pieza4------------------------------------------------------------------
#RobotA se acerca a la MesaA1
ap4=transl(1323.030,-411.739,93.068)*roty(pi)           #Se cambia el AproxMesaA1_P__________________________
robotA.MoveJ(ap4)
robotA.setSpeed(1000)
#RobotA toma la pieza4 de la MesaA1
bp4=transl(1323.030,-410.438,-220.350)*roty(pi)        #Se cambia respecto a Left_P________________________
robotA.MoveJ(bp4)
robotA.setSpeed(1000)
mesafinal.DetachAll()
pi4.setParentStatic(gripper1)
#RobotA se aleja de la MesaA1
cp4=transl(1323.030,-411.739,93.068)*roty(pi)           #Se cambia el AproxMesaA1_P__________________________
robotA.MoveJ(cp4)
robotA.setSpeed(1000)
#RobotA se aproxima a MesaA0 para dejar la pieza
dp4= transl(1323.030,430.867,93.068)*roty(pi)      #Se cambia respecto a AproxMesaA0_P________________________
robotA.MoveJ(dp4)
robotA.setSpeed(1000)
#RobotA deja la pieza4 de la MesaA0
ep4= transl(1323.030,430.867,-220.350)*roty(pi)    #Se cambia respecto a Take_P________________________
robotA.MoveJ(ep4)
robotA.setSpeed(1000)
gripper1.DetachAll()                      #Se cambia el pi_____________________________________
#RobotA se mueve a la posición de home
fp4=transl(945.000,0.000,834.135)*roty(pi)
robotA.MoveJ(fp4)
robotA.setSpeed(1000)

#Colocando a posición inicial Pieza5------------------------------------------------------------------
#RobotA se acerca a la MesaA1
ap5=transl(1323.030,-237.214,93.068)*roty(pi)           #Se cambia el AproxMesaA1_P__________________________
robotA.MoveJ(ap5)
robotA.setSpeed(1000)
#RobotA toma la pieza5 en la MesaA1
bp5=transl(1323.030,-235.913,-220.350)*roty(pi)        #Se cambia respecto a Left_P________________________
robotA.MoveJ(bp5)
robotA.setSpeed(1000)
mesafinal.DetachAll()
pi5.setParentStatic(gripper1)
#RobotA se aleja de la MesaA1
cp5=transl(1323.030,-237.214,93.068)*roty(pi)           #Se cambia el AproxMesaA1_P__________________________
robotA.MoveJ(cp5)
robotA.setSpeed(1000)
#RobotA se aproxima a MesaA0 para dejar la pieza
dp5= transl(1323.030,257.289,93.068)*roty(pi)      #Se cambia respecto a AproxMesaA0_P________________________
robotA.MoveJ(dp5)
robotA.setSpeed(1000)
#RobotA deja la pieza5 en la MesaA0
ep5= transl(1323.030,257.289,-220.350)*roty(pi)    #Se cambia respecto a Take_P________________________
robotA.MoveJ(ep5)
robotA.setSpeed(1000)
gripper1.DetachAll()                      #Se cambia el pi_____________________________________
#RobotA se mueve a la posición de home
fp5=transl(945.000,0.000,834.135)*roty(pi)
robotA.MoveJ(fp5)
robotA.setSpeed(1000)
